(* POU FB_BACnet_AnalogOutput_EX, ST *)
FUNCTION_BLOCK FB_BACnet_AnalogOutput_EX
VAR_INPUT
	bEnablePV			: BOOL; (* enable present value with priority x in priority array, FALSE = priority x disable *)
	bNullPV				: BOOL; (* clear priority entry *)
	fPV					: REAL; (* decimal number for priority x, when input bEnablePV is TRUE *)
END_VAR
VAR_IN_OUT
	Device				: FB_BACnet_Device;
END_VAR
VAR_OUTPUT
	bReady				: BOOL;
	fPresentValue		: REAL;
	bOverridden			: BOOL;
	bOutOfService		: BOOL;
	bFault				: BOOL;
	bInAlarm			: BOOL;
	bNoOutput			: BOOL;
	bOpenLoop			: BOOL;
	bShortedLoop		: BOOL;
	bOtherFault			: BOOL;
	eEventState			: E_BACNETEVENTSTATE;
	bAckedTrans_ToOffNormal : BOOL;
	bAckedTrans_ToFault		: BOOL;
	bAckedTrans_ToNormal	: BOOL;
	nActivePrio			: UINT;
	tObjectID			: T_BACnet_ObjectIdentifier := 16#FFFFFFFF;
	bError				: BOOL;
	nErrorId			: UINT;
END_VAR
VAR
	_PresentValue AT%I*: REAL; 			(* ~(BACnet_PresentValue 			:		: )
								   			(BACnet_ObjectType 				: AO	: )	*)
    _PresentValue_Priority12 AT%Q*: DWORD;(* ~(BACnet_PresentValue_Priority12:		: )	*)
	_ActivePriority AT%I*: UDINT; 		(* ~(BACnet_ActivePriority 			:		: )	*)
	_ObjectId AT%I*: DWORD;				(* ~(BACnet_ObjectIdentifier		:		: LINK) *)
	_StatusFlags AT%I*: WORD; 			(* ~(BACnet_StatusFlags 			:		: )	*)
	_EventState AT%I*: WORD;			(* ~(BACnet_EventState 				:		: )	*)
	_Reliability AT%I*: WORD; 			(* ~(BACnet_Reliability 			:		: )	*)
	_AckedTransitions AT%I*:WORD;		(* ~(BACnet_AckedTransitions		:		: ) *)
	_StatusFlagsBits : ST_BACnet_StatusFlags;
	_AckedTransBits : ST_BACnet_EventTransitionBits;
	_nUpdateCount : UDINT := 0;
END_VAR
(* update server device *)
IF (Device._nUpdateCount = _nUpdateCount) THEN
	Device();
END_IF
(* remind current number of update counter *)
_nUpdateCount := Device._nUpdateCount;

IF Device.bFirstCycle THEN
	(* first call of the server device since reboot/reset *)
	bReady := FALSE;
	_PresentValue_Priority12 := F_BACnet_RealNothing();

ELSIF (F_BACnet_GetObjType(_ObjectId) <> BACnetObjectType_AnalogOutput) THEN
	(* wrong mapping / invalid object ID *)
	IF _ObjectId = 0 THEN
		nErrorId := BACnet_ERR_WRONG_MAPPING;
	ELSE
		nErrorId := BACnet_ERR_INVALID_OBJECTID;
	END_IF
	bReady := FALSE;

ELSIF (_StatusFlags < 4) THEN
	(* wrong mapping *)
	nErrorId := BACnet_ERR_WRONG_MAPPING;
	bReady := FALSE;

ELSIF Device.bOperational THEN
	(* ready state *)
	bReady := TRUE;
	nErrorId := BACnet_ERR_NO_ERROR;

	(* write into priority array *)
	_PresentValue_Priority12 := F_BACnet_RealPV(bEnablePV, bNullPV, fPV);

	(* present value *)
	fPresentValue := _PresentValue;

	(* build bit states *)
	_StatusFlagsBits := F_BACnet_StatusFlags(_StatusFlags);
	_AckedTransBits		:= F_BACnet_EventTransitionFlags(_AckedTransitions);

	(* copy states to output *)
	bOverridden := _StatusFlagsBits.overridden;
	bOutOfService := _StatusFlagsBits.out_of_service;
	bFault := _StatusFlagsBits.fault;
	bInAlarm := _StatusFlagsBits.in_alarm;
	bNoOutput := (_Reliability = BACnetReliability_no_output);
	bOpenLoop := (_Reliability = BACnetReliability_open_loop);
	bShortedLoop := (_Reliability = BACnetReliability_shorted_loop);
	bOtherFault := (_Reliability = BACnetReliability_unreliable_other);
	bAckedTrans_ToOffNormal := _AckedTransBits.to_offnormal;
	bAckedTrans_ToFault := _AckedTransBits.to_fault;
	bAckedTrans_ToNormal := _AckedTransBits.to_normal;
	tObjectID := _ObjectId;

	(* convert enumeration *)
	eEventState := _EventState;

	(* copy active priority *)
	nActivePrio := UDINT_TO_UINT(_ActivePriority);

ELSE
	(* server device not ready, reset local ready also *)
	bReady := FALSE;
	nErrorId := BACnet_ERR_OPERATIONAL;
END_IF
(* set error flag *)
bError := (nErrorId <> BACnet_ERR_NO_ERROR);
END_FUNCTION_BLOCK

(* POU FB_BACnet_AnalogOutput_RAW, ST *)
FUNCTION_BLOCK FB_BACnet_AnalogOutput_RAW
VAR_INPUT
	bEnablePV		: BOOL; (* enable present value with priority x in priority array, FALSE = priority x disable *)
	bNullPV			: BOOL; (* clear priority entry *)
	fPV				: REAL; (* decimal number for priority x, when input bEnablePV is TRUE *)
	bRawOverridden	AT%Q*: BOOL; (* ~(BACnet_RawIoStateOverride	:		: ) *)
	bNoOutput		: BOOL;
	bOpenLoop		: BOOL;
	bShortedLoop	: BOOL;
	bCommFailure	: BOOL;
	bOtherFault		: BOOL;
END_VAR
VAR_IN_OUT
	Device	: FB_BACnet_Device;
END_VAR
VAR_OUTPUT
	bReady			: BOOL;
	fPresentValue	: REAL;
	bOverridden		: BOOL;
	bOutOfService	: BOOL;
	bFault			: BOOL;
	bInAlarm		: BOOL;
	bAckedTrans_ToOffNormal : BOOL;
	bAckedTrans_ToFault		: BOOL;
	bAckedTrans_ToNormal	: BOOL;
	bError			: BOOL;
	nErrorId		: UINT;
	nRawOut			AT%I*: INT;			(* ~(BACnet_RawIoAnalogSignedValue : : ) *)
END_VAR
VAR
	_PresentValue AT%I*: REAL; 			(* ~(BACnet_PresentValue 			:		: )
								   			(BACnet_ObjectType 				: AO	: )	*)
	_ObjectId AT%I*: DWORD;				(* ~(BACnet_ObjectIdentifier		:		: LINK) *)
	_AckedTransitions AT%I*:WORD;		(* ~(BACnet_AckedTransitions		:		: ) *)
	_StatusFlags AT%I*: WORD; 			(* ~(BACnet_StatusFlags 			:		: )	*)
    _PresentValue_Priority12 AT%Q*: DWORD;(* ~(BACnet_PresentValue_Priority12:		: )	*)
	_Reliability AT%Q*: WORD := BACnetReliability_no_fault_detected;(* ~(BACnet_Reliability 	:		: )	*)
	_AckedTransBits : ST_BACnet_EventTransitionBits;
	_StatusFlagsBits : ST_BACnet_StatusFlags;
	_nUpdateCount : UDINT := 0;
END_VAR
(* update server device *)
IF (Device._nUpdateCount = _nUpdateCount) THEN
	Device();
END_IF
(* remind current number of update counter *)
_nUpdateCount := Device._nUpdateCount;

(* handle raw error *)
IF bNoOutput THEN
	_Reliability := BACnetReliability_no_output;
ELSIF bOpenLoop THEN
	_Reliability := BACnetReliability_open_loop;
ELSIF bShortedLoop THEN
	_Reliability := BACnetReliability_shorted_loop;
ELSIF bCommFailure THEN
	_Reliability := BACnetReliability_communication_failure;
ELSIF bOtherFault THEN
	_Reliability := BACnetReliability_unreliable_other;
ELSE
	_Reliability := BACnetReliability_no_fault_detected;
END_IF

IF Device.bFirstCycle THEN
	(* first call of the server device since reboot/reset *)
	bReady := FALSE;
	_PresentValue_Priority12 := F_BACnet_RealNothing();

ELSIF (_StatusFlags < 4) THEN
	(* wrong mapping *)
	nErrorId := BACnet_ERR_WRONG_MAPPING;
	bReady := FALSE;

ELSIF Device.bOperational THEN
	(* ready state *)
	bReady := TRUE;
	nErrorId := BACnet_ERR_NO_ERROR;

	(* write into priority array *)
	_PresentValue_Priority12 := F_BACnet_RealPV(bEnablePV, bNullPV, fPV);

	(* present value *)
	fPresentValue := _PresentValue;

	(* build bit states *)
	_StatusFlagsBits := F_BACnet_StatusFlags(_StatusFlags);
	_AckedTransBits		:= F_BACnet_EventTransitionFlags(_AckedTransitions);

	(* copy states to output *)
	bOverridden := _StatusFlagsBits.overridden;
	bOutOfService := _StatusFlagsBits.out_of_service;
	bFault := _StatusFlagsBits.fault;
	bInAlarm := _StatusFlagsBits.in_alarm;
	bAckedTrans_ToOffNormal := _AckedTransBits.to_offnormal;
	bAckedTrans_ToFault := _AckedTransBits.to_fault;
	bAckedTrans_ToNormal := _AckedTransBits.to_normal;

ELSE
	(* server device not ready, reset local ready also *)
	bReady := FALSE;
	nErrorId := BACnet_ERR_OPERATIONAL;
END_IF
(* set error flag *)
bError := (nErrorId <> BACnet_ERR_NO_ERROR);
END_FUNCTION_BLOCK

(* POU FB_BACnet_AnalogValue, ST *)
FUNCTION_BLOCK FB_BACnet_AnalogValue
VAR_INPUT
	bEnablePV		: BOOL; (* enable present value with priority x in priority array, FALSE = priority x disable *)
	bNullPV			: BOOL; (* clear priority entry *)
	fPV				: REAL; (* decimal number for priority x, when input bEnablePV is TRUE *)
END_VAR
VAR_IN_OUT
	Device			: FB_BACnet_Device;
END_VAR
VAR_OUTPUT
	bReady			: BOOL;
	fPresentValue	: REAL;
	bOverridden		: BOOL;
	bOutOfService	: BOOL;
	bFault			: BOOL;
	bInAlarm		: BOOL;
	bError			: BOOL;
	nErrorId		: UINT;
END_VAR
VAR
	_PresentValue AT%I*: REAL; 			(* ~(BACnet_PresentValue 			:		: )
								   			(BACnet_ObjectType 				: AV	: )	*)
    _PresentValue_Priority12 AT%Q*: DWORD;(* ~(BACnet_PresentValue_Priority12:		: )	*)
	_StatusFlags AT%I*: WORD; 			(* ~(BACnet_StatusFlags 			:		: )	*)
	_StatusFlagsBits : ST_BACnet_StatusFlags;
	_nUpdateCount : UDINT := 0;
END_VAR
(* update server device *)
IF (Device._nUpdateCount = _nUpdateCount) THEN
	Device();
END_IF
(* remind current number of update counter *)
_nUpdateCount := Device._nUpdateCount;

IF Device.bFirstCycle THEN
	(* first call of the server device since reboot/reset *)
	bReady := FALSE;
	_PresentValue_Priority12 := F_BACnet_RealNothing();
ELSIF (_StatusFlags < 4) THEN
	(* wrong mapping *)
	nErrorId := BACnet_ERR_WRONG_MAPPING;
	bReady := FALSE;

ELSIF Device.bOperational THEN
	(* ready state *)
	bReady := TRUE;
	nErrorId := BACnet_ERR_NO_ERROR;

	(* write into priority array *)
	_PresentValue_Priority12 := F_BACnet_RealPV(bEnablePV, bNullPV, fPV);

	(* present value *)
	fPresentValue := _PresentValue;

	(* build bit states *)
	_StatusFlagsBits := F_BACnet_StatusFlags(_StatusFlags);

	(* copy states to output *)
	bOverridden := _StatusFlagsBits.overridden;
	bOutOfService := _StatusFlagsBits.out_of_service;
	bFault := _StatusFlagsBits.fault;
	bInAlarm := _StatusFlagsBits.in_alarm;

ELSE
	(* server device not ready, reset local ready also *)
	bReady := FALSE;
	nErrorId := BACnet_ERR_OPERATIONAL;
END_IF
(* set error flag *)
bError := (nErrorId <> BACnet_ERR_NO_ERROR);
END_FUNCTION_BLOCK

(* POU FB_BACnet_AnalogValue_ADS, ST *)
FUNCTION_BLOCK FB_BACnet_AnalogValue_ADS
VAR_INPUT
	bEnablePV			: BOOL; (* enable PV write commands *)
	bNullPV				: BOOL; (* clear priority entry *)
	fPV					: REAL; (* decimal number for priority x, when input bEnablePV is TRUE and bNullPV is FALSE *)
	bManual				: BOOL; (* FALSE --> TRUE: write present_value immediately, FALSE: only write present_value on-change, TRUE: write present_value on-change and when device turns operational *)
	ePriority			: E_BACNETPRIORITY := BACNETPRIORITY_12;
END_VAR
VAR_IN_OUT
	Device				: FB_BACnet_Device;
END_VAR
VAR_OUTPUT
	bReady				: BOOL;
	bPvDone				: BOOL; (* present_value written over ADS *)
	fPresentValue		: REAL;
	bOverridden			: BOOL;
	bOutOfService		: BOOL;
	bFault				: BOOL;
	bInAlarm			: BOOL;
	tObjectID			: T_BACnet_ObjectIdentifier := 16#FFFFFFFF;
	bError				: BOOL;
	nErrorId			: UINT;
	nAdsErrorId			: UDINT;
END_VAR
VAR
	_PresentValue AT%I*: REAL; 			(* ~(BACnet_PresentValue 		:		: )
								   			(BACnet_ObjectType 			: AV	: )	*)
	_ObjectId AT%I*: DWORD;				(* ~(BACnet_ObjectIdentifier	:		: LINK) *)
	_StatusFlags AT%I*: WORD; 			(* ~(BACnet_StatusFlags 		:		: )	*)
    _PresentValue_Ads : DWORD;
	_StatusFlagsBits : ST_BACnet_StatusFlags;
	_nUpdateCount : UDINT := 0;
	_WriteProp : FB_BACnet_WriteProp;
	_rtrigManual : R_TRIG;
	_bNullPvOld : BOOL;
	_nObjType : E_BACNETOBJECTTYPE;
END_VAR
(* update server device *)
IF (Device._nUpdateCount = _nUpdateCount) THEN
	Device();
END_IF
(* remind current number of update counter *)
_nUpdateCount := Device._nUpdateCount;

(* trigger on manual flag *)
_rtrigManual(CLK:= bManual, Q=> );

(* decode object type *)
_nObjType := F_BACnet_GetObjType(_ObjectId);

IF Device.bFirstCycle THEN
	(* first call of the server device since reboot/reset *)
	bReady := FALSE;
	bPvDone := FALSE;

ELSIF _nObjType <> BACnetObjectType_AnalogValue THEN
	(* wrong mapped object type *)
	nErrorId := BACnet_ERR_INVALID_OBJECTTYPE;
	bReady := FALSE;
	bPvDone := FALSE;

ELSIF (_StatusFlags < 4) THEN
	(* wrong mapping *)
	nErrorId := BACnet_ERR_WRONG_MAPPING;
	bReady := FALSE;
	bPvDone := FALSE;

ELSIF Device.bOperational THEN

	IF Device.stAdsConn.bValid THEN
		(* write present_value on manual trigger, on-change and on operational recover *)
		IF		bEnablePV
			AND	(		_rtrigManual.Q
					OR	(MEMCMP(pBuf1:=ADR(fPV), pBuf2:=ADR(_PresentValue_Ads), n:=SIZEOF(_PresentValue_Ads)) <> 0)
					OR	((NOT bReady) AND bManual)
					OR	(bNullPV <> _bNullPvOld)
				)
		THEN
			_WriteProp.bExecute := TRUE;
			bPvDone := FALSE;
			(* write depending on enable state *)
			_PresentValue_Ads := F_BACnet_RealPV(TRUE, bNullPV, fPV);
			(* remind null flag *)
			_bNullPvOld := bNullPV;
		END_IF

		(* ready state *)
		IF (nAdsErrorId = 0) THEN
			bReady := TRUE;
			nErrorId := BACnet_ERR_NO_ERROR;
		END_IF

	ELSE
		(* invalid ADS connection *)
		bReady := FALSE;
		nErrorId := BACnet_ERR_INVALID_ADS_CONN;
		bPvDone := FALSE;
	END_IF

	(* present value *)
	fPresentValue := _PresentValue;

	(* build bit states *)
	_StatusFlagsBits := F_BACnet_StatusFlags(_StatusFlags);

	(* copy states to output *)
	bOverridden := _StatusFlagsBits.overridden;
	bOutOfService := _StatusFlagsBits.out_of_service;
	bFault := _StatusFlagsBits.fault;
	bInAlarm := _StatusFlagsBits.in_alarm;
	tObjectID := _ObjectId;

ELSE
	(* server device not ready, reset local ready also *)
	bReady := FALSE;
	nErrorId := BACnet_ERR_OPERATIONAL;
	bPvDone := FALSE;
END_IF

(* call write property command *)
_WriteProp(
	BACnetDevicePort	:= Device.stAdsConn.nAmsPort,
	bExecute			:= ,
	sNetId				:= Device.stAdsConn.sAmsNetId,
	ObjectType			:= _nObjType,
	PropertyID			:= BACnetPropertyIdentifier_PresentValue,
	Priority			:= ePriority,
	DataType			:= BACnetDataType_Real,
	ObjectInstance		:= F_BACnet_GetObjInstance(_ObjectId),
	ptrValue			:= ADR(_PresentValue_Ads),
	nLenValue			:= SIZEOF(_PresentValue_Ads),
	bDone				=> ,
	bBusy				=> ,
	bError				=> ,
	nErrID				=> );

(* set done flag *)
IF _WriteProp.bExecute AND (NOT _WriteProp.bBusy) THEN
	(* check if command was finished with error *)
	IF _WriteProp.bError THEN
		bPvDone		:= FALSE;
		bReady		:= FALSE;
		nErrorId	:= BACnet_ERR_ADS_Write;
	ELSE
		(* successful written *)
		bPvDone		:= TRUE;
	END_IF
	nAdsErrorId := _WriteProp.nErrID;
	(* reset execution bit *)
	_WriteProp(bExecute := FALSE);
END_IF

(* set error flag *)
bError := (nErrorId <> BACnet_ERR_NO_ERROR) OR (nAdsErrorId <> 0);
END_FUNCTION_BLOCK

(* POU FB_BACnet_AnalogValue_EX, ST *)
FUNCTION_BLOCK FB_BACnet_AnalogValue_EX
VAR_INPUT
	bEnablePV			: BOOL; (* enable present value with priority x in priority array, FALSE = priority x disable *)
	bNullPV				: BOOL; (* clear priority entry *)
	fPV					: REAL; (* decimal number for priority x, when input bEnablePV is TRUE *)
END_VAR
VAR_IN_OUT
	Device				: FB_BACnet_Device;
END_VAR
VAR_OUTPUT
	bReady				: BOOL;
	fPresentValue		: REAL;
	bOverridden			: BOOL;
	bOutOfService		: BOOL;
	bFault				: BOOL;
	bInAlarm			: BOOL;
	bOverRange			: BOOL;
	bUnderRange			: BOOL;
	bOtherFault			: BOOL;
	eEventState			: E_BACNETEVENTSTATE;
	bAckedTrans_ToOffNormal : BOOL;
	bAckedTrans_ToFault		: BOOL;
	bAckedTrans_ToNormal	: BOOL;
	nActivePrio			: UINT;
	tObjectID			: T_BACnet_ObjectIdentifier := 16#FFFFFFFF;
	bError				: BOOL;
	nErrorId			: UINT;
END_VAR
VAR
	_PresentValue AT%I*: REAL; 			(* ~(BACnet_PresentValue 				:		: )
								   			(BACnet_ObjectType 					: AV	: )	*)
    _PresentValue_Priority12 AT%Q*: DWORD;(* ~(BACnet_PresentValue_Priority12	:		: )	*)
	_ActivePriority AT%I*: UDINT; 		(* ~(BACnet_ActivePriority 				:		: )	*)
	_ObjectId AT%I*: DWORD;				(* ~(BACnet_ObjectIdentifier			:		: LINK) *)
	_StatusFlags AT%I*: WORD; 			(* ~(BACnet_StatusFlags 				:		: )	*)
	_EventState AT%I*: WORD;			(* ~(BACnet_EventState 					:		: )	*)
	_Reliability AT%I*: WORD;			(* ~(BACnet_Reliability 				:		: )	*)
	_AckedTransitions AT%I*:WORD;		(* ~(BACnet_AckedTransitions			:		: ) *)
	_StatusFlagsBits : ST_BACnet_StatusFlags;
	_AckedTransBits : ST_BACnet_EventTransitionBits;
	_nUpdateCount : UDINT := 0;
END_VAR
(* update server device *)
IF (Device._nUpdateCount = _nUpdateCount) THEN
	Device();
END_IF
(* remind current number of update counter *)
_nUpdateCount := Device._nUpdateCount;

IF Device.bFirstCycle THEN
	(* first call of the server device since reboot/reset *)
	bReady := FALSE;
	_PresentValue_Priority12 := F_BACnet_RealNothing();

ELSIF (F_BACnet_GetObjType(_ObjectId) <> BACnetObjectType_AnalogValue) THEN
	(* wrong mapping / invalid object ID *)
	IF _ObjectId = 0 THEN
		nErrorId := BACnet_ERR_WRONG_MAPPING;
	ELSE
		nErrorId := BACnet_ERR_INVALID_OBJECTID;
	END_IF
	bReady := FALSE;

ELSIF (_StatusFlags < 4) THEN
	(* wrong mapping *)
	nErrorId := BACnet_ERR_WRONG_MAPPING;
	bReady := FALSE;

ELSIF Device.bOperational THEN
	(* ready state *)
	bReady := TRUE;
	nErrorId := BACnet_ERR_NO_ERROR;

	(* write into priority array *)
	_PresentValue_Priority12 := F_BACnet_RealPV(bEnablePV, bNullPV, fPV);

	(* present value *)
	fPresentValue := _PresentValue;

	(* build bit states *)
	_StatusFlagsBits := F_BACnet_StatusFlags(_StatusFlags);
	_AckedTransBits		:= F_BACnet_EventTransitionFlags(_AckedTransitions);

	(* copy states to output *)
	bOverridden := _StatusFlagsBits.overridden;
	bOutOfService := _StatusFlagsBits.out_of_service;
	bFault := _StatusFlagsBits.fault;
	bInAlarm := _StatusFlagsBits.in_alarm;
	bOverRange := (_Reliability = BACnetReliability_over_range);
	bUnderRange := (_Reliability = BACnetReliability_under_range);
	bOtherFault := (_Reliability = BACnetReliability_unreliable_other);
	bAckedTrans_ToOffNormal := _AckedTransBits.to_offnormal;
	bAckedTrans_ToFault := _AckedTransBits.to_fault;
	bAckedTrans_ToNormal := _AckedTransBits.to_normal;
	tObjectID := _ObjectId;

	(* convert enumeration *)
	eEventState := _EventState;

	(* copy active priority *)
	nActivePrio := UDINT_TO_UINT(_ActivePriority);
ELSE
	(* server device not ready, reset local ready also *)
	bReady := FALSE;
	nErrorId := BACnet_ERR_OPERATIONAL;
END_IF
(* set error flag *)
bError := (nErrorId <> BACnet_ERR_NO_ERROR);
END_FUNCTION_BLOCK

(* POU FB_BACnet_Averaging, ST *)
FUNCTION_BLOCK FB_BACnet_Averaging
VAR_IN_OUT
	Device			: FB_BACnet_Device;
END_VAR
VAR_OUTPUT
	bReady			: BOOL;
	fAverageValue	: REAL;
	fMaximumValue	: REAL;
	fMinimumValue	: REAL;
	nValidSamples	: UDINT;
	nWindowSamples	: UDINT;
	nWindowInterval	: UDINT; (* [s] *)
	bError			: BOOL;
	nErrorId		: UINT;
END_VAR
VAR
	_AverageValue AT%I*: REAL;			(* ~(BACnet_AverageValue	:		: )
											(BACnet_ObjectType 		: AVG	: ) *)
	_MaximumValue AT%I*: REAL;			(* ~(BACnet_MaximumValue	:		: ) *)
	_MinimumValue AT%I*: REAL;			(* ~(BACnet_MinimumValue	:		: ) *)
	_ValidSamples AT%I*: UDINT;			(* ~(BACnet_ValidSamples	:		: ) *)
	_WindowSamples AT%I*: UDINT;		(* ~(BACnet_WindowSamples	:		: ) *)
	_WindowInterval AT%I*: UDINT;		(* ~(BACnet_WindowInterval	:		: ) *)
	_nUpdateCount : UDINT := 0;
END_VAR
(* update server device *)
IF (Device._nUpdateCount = _nUpdateCount) THEN
	Device();
END_IF
(* remind current number of update counter *)
_nUpdateCount := Device._nUpdateCount;

IF Device.bFirstCycle THEN
	(* first call of the server device since reboot/reset *)
	bReady := FALSE;
ELSIF Device.bOperational THEN
	(* ready state *)
	bReady := TRUE;
	nErrorId := BACnet_ERR_NO_ERROR;

	(* present values *)
	fAverageValue	:= _AverageValue;
	fMaximumValue	:= _MaximumValue;
	fMinimumValue	:= _MinimumValue;
	nValidSamples	:= _ValidSamples;
	nWindowSamples	:= _WindowSamples;
	nWindowInterval	:= _WindowInterval;

ELSE
	(* server device not ready, reset local ready also *)
	bReady := FALSE;
	nErrorId := BACnet_ERR_OPERATIONAL;
END_IF
(* set error flag *)
bError := (nErrorId <> BACnet_ERR_NO_ERROR);
END_FUNCTION_BLOCK

(* POU FB_BACnet_Averaging_EX, ST *)
FUNCTION_BLOCK FB_BACnet_Averaging_EX
VAR_IN_OUT
	Device				: FB_BACnet_Device;
END_VAR
VAR_OUTPUT
	bReady				: BOOL;
	fAverageValue		: REAL;
	fMaximumValue		: REAL;
	fMinimumValue		: REAL;
	nValidSamples		: UDINT;
	nWindowSamples		: UDINT;
	nWindowInterval		: UDINT; (* [s] *)
	tObjectID			: T_BACnet_ObjectIdentifier := 16#FFFFFFFF;
	bError				: BOOL;
	nErrorId			: UINT;
END_VAR
VAR
	_AverageValue AT%I*: REAL;			(* ~(BACnet_AverageValue	:		: )
											(BACnet_ObjectType 		: AVG	: ) *)
	_MaximumValue AT%I*: REAL;			(* ~(BACnet_MaximumValue	:		: ) *)
	_MinimumValue AT%I*: REAL;			(* ~(BACnet_MinimumValue	:		: ) *)
	_ValidSamples AT%I*: UDINT;			(* ~(BACnet_ValidSamples	:		: ) *)
	_WindowSamples AT%I*: UDINT;		(* ~(BACnet_WindowSamples	:		: ) *)
	_WindowInterval AT%I*: UDINT;		(* ~(BACnet_WindowInterval	:		: ) *)
	_ObjectId AT%I*: DWORD;				(* ~(BACnet_ObjectIdentifier:		: LINK) *)
	_nUpdateCount : UDINT := 0;
END_VAR
(* update server device *)
IF (Device._nUpdateCount = _nUpdateCount) THEN
	Device();
END_IF
(* remind current number of update counter *)
_nUpdateCount := Device._nUpdateCount;

IF Device.bFirstCycle THEN
	(* first call of the server device since reboot/reset *)
	bReady := FALSE;

ELSIF (F_BACnet_GetObjType(_ObjectId) <> BACnetObjectType_Averaging) THEN
	(* wrong mapping / invalid object ID *)
	IF _ObjectId = 0 THEN
		nErrorId := BACnet_ERR_WRONG_MAPPING;
	ELSE
		nErrorId := BACnet_ERR_INVALID_OBJECTID;
	END_IF
	bReady := FALSE;
	tObjectID := 16#FFFFFFFF;

ELSIF Device.bOperational THEN
	(* ready state *)
	bReady := TRUE;
	nErrorId := BACnet_ERR_NO_ERROR;

	(* present values *)
	fAverageValue	:= _AverageValue;
	fMaximumValue	:= _MaximumValue;
	fMinimumValue	:= _MinimumValue;
	nValidSamples	:= _ValidSamples;
	nWindowSamples	:= _WindowSamples;
	nWindowInterval	:= _WindowInterval;

	(* other states *)
	tObjectID := _ObjectId;

ELSE
	(* server device not ready, reset local ready also *)
	bReady := FALSE;
	nErrorId := BACnet_ERR_OPERATIONAL;
END_IF
(* set error flag *)
bError := (nErrorId <> BACnet_ERR_NO_ERROR);
END_FUNCTION_BLOCK

(* POU FB_BACnet_BinaryInput, ST *)
FUNCTION_BLOCK FB_BACnet_BinaryInput
VAR_IN_OUT
	Device	: FB_BACnet_Device;
END_VAR
VAR_OUTPUT
	bReady			: BOOL;
	bPresentValue	: BOOL;
	bOverridden		: BOOL;
	bOutOfService	: BOOL;
	bFault			: BOOL;
	bInAlarm		: BOOL;
	bError			: BOOL;
	nErrorId		: UINT;
END_VAR
VAR
	_PresentValue AT%I*: WORD; 			(* ~(BACnet_PresentValue 		:		: )
											(BACnet_ObjectType			:BI    	: )	*)
	_StatusFlags AT%I*: WORD; 			(* ~(BACnet_StatusFlags 		:	    : )	*)
	_StatusFlagsBits : ST_BACnet_StatusFlags;
	_nUpdateCount : UDINT := 0;
END_VAR
(* update server device *)
IF (Device._nUpdateCount = _nUpdateCount) THEN
	Device();
END_IF
(* remind current number of update counter *)
_nUpdateCount := Device._nUpdateCount;

(* check BitString format of StatusFlags --> if StatusFlags are less than 4, object isn't linked correctly *)
IF (_StatusFlags < 4) THEN
	(* wrong mapping *)
	nErrorId := BACnet_ERR_WRONG_MAPPING;
	bReady := FALSE;

ELSIF Device.bOperational THEN
	(* ready state *)
	bReady := TRUE;
	nErrorId := BACnet_ERR_NO_ERROR;

	(* present value *)
	bPresentValue := F_BinPV_To_Bool(_PresentValue);

	(* build bit states *)
	_StatusFlagsBits := F_BACnet_StatusFlags(_StatusFlags);

	(* copy states to output *)
	bOverridden := _StatusFlagsBits.overridden;
	bOutOfService := _StatusFlagsBits.out_of_service;
	bFault := _StatusFlagsBits.fault;
	bInAlarm := _StatusFlagsBits.in_alarm;

ELSE
	bReady := FALSE;
	nErrorId := BACnet_ERR_OPERATIONAL;
END_IF
(* set error flag *)
bError := (nErrorId <> BACnet_ERR_NO_ERROR);
END_FUNCTION_BLOCK

(* POU FB_BACnet_BinaryInput_EX, ST *)
FUNCTION_BLOCK FB_BACnet_BinaryInput_EX
VAR_IN_OUT
	Device	: FB_BACnet_Device;
END_VAR
VAR_OUTPUT
	bReady				: BOOL;
	bPresentValue		: BOOL;
	bOverridden			: BOOL;
	bOutOfService		: BOOL;
	bFault				: BOOL;
	bInAlarm			: BOOL;
	bNoSensor			: BOOL;
	bOpenLoop			: BOOL;
	bShortedLoop		: BOOL;
	bOtherFault			: BOOL;
	eEventState			: E_BACNETEVENTSTATE;
	bAckedTrans_ToOffNormal : BOOL;
	bAckedTrans_ToFault		: BOOL;
	bAckedTrans_ToNormal	: BOOL;
	nChangeOfState		: UDINT;
	tObjectID			: T_BACnet_ObjectIdentifier := 16#FFFFFFFF;
	bError				: BOOL;
	nErrorId			: UINT;
END_VAR
VAR
	_ChangeOfStateCount AT%I*: UDINT;		(* ~(BACnet_ChangeOfStateCount	:		: ) *)
	_ObjectId AT%I*: DWORD;					(* ~(BACnet_ObjectIdentifier	:		: LINK) *)
	_PresentValue AT%I*: WORD; 				(* ~(BACnet_PresentValue 		:		: )
												(BACnet_ObjectType			:BI    	: )	*)
	_StatusFlags AT%I*: WORD; 				(* ~(BACnet_StatusFlags 		:	    : )	*)
	_EventState AT%I*: WORD; 				(* ~(BACnet_EventState 			:	    : )	*)
	_Reliability AT%I*: WORD; 				(* ~(BACnet_Reliability 		:		: )	*)
	_AckedTransitions AT%I*:WORD;			(* ~(BACnet_AckedTransitions	:		: ) *)
	_AckedTransBits : ST_BACnet_EventTransitionBits;
	_StatusFlagsBits : ST_BACnet_StatusFlags;
	_nUpdateCount : UDINT := 0;
END_VAR
(* update server device *)
IF (Device._nUpdateCount = _nUpdateCount) THEN
	Device();
END_IF
(* remind current number of update counter *)
_nUpdateCount := Device._nUpdateCount;

(* check object type *)
IF (F_BACnet_GetObjType(_ObjectId) <> BACnetObjectType_BinaryInput) THEN
	(* wrong mapping / invalid object ID *)
	IF _ObjectId = 0 THEN
		nErrorId := BACnet_ERR_WRONG_MAPPING;
	ELSE
		nErrorId := BACnet_ERR_INVALID_OBJECTID;
	END_IF
	bReady := FALSE;

ELSIF (_StatusFlags < 4) THEN
	(* wrong mapping *)
	nErrorId := BACnet_ERR_WRONG_MAPPING;
	bReady := FALSE;

ELSIF Device.bOperational THEN
	(* ready state *)
	bReady := TRUE;
	nErrorId := BACnet_ERR_NO_ERROR;

	(* present value *)
	bPresentValue := F_BinPV_To_Bool(_PresentValue);

	(* build bit states *)
	_StatusFlagsBits := F_BACnet_StatusFlags(_StatusFlags);
	_AckedTransBits		:= F_BACnet_EventTransitionFlags(_AckedTransitions);

	(* copy states to output *)
	bOverridden := _StatusFlagsBits.overridden;
	bOutOfService := _StatusFlagsBits.out_of_service;
	bFault := _StatusFlagsBits.fault;
	bInAlarm := _StatusFlagsBits.in_alarm;
	bNoSensor := (_Reliability = BACnetReliability_no_sensor);
	bOpenLoop := (_Reliability = BACnetReliability_open_loop);
	bShortedLoop := (_Reliability = BACnetReliability_shorted_loop);
	bOtherFault := (_Reliability = BACnetReliability_unreliable_other);
	bAckedTrans_ToOffNormal := _AckedTransBits.to_offnormal;
	bAckedTrans_ToFault := _AckedTransBits.to_fault;
	bAckedTrans_ToNormal := _AckedTransBits.to_normal;
	tObjectID := _ObjectId;

	(* convert enumeration *)
	eEventState := _EventState;

	(* copy change_of_state_count *)
	nChangeOfState := _ChangeOfStateCount;
ELSE
	bReady := FALSE;
	nErrorId := BACnet_ERR_OPERATIONAL;
END_IF
(* set error flag *)
bError := (nErrorId <> BACnet_ERR_NO_ERROR);
END_FUNCTION_BLOCK

(* POU FB_BACnet_BinaryInput_RAW, ST *)
FUNCTION_BLOCK FB_BACnet_BinaryInput_RAW
VAR_INPUT
	bRawIn			AT%Q*: BOOL; (* ~(BACnet_RawIoBinaryBoolValue : : ) *)
	bNoSensor		: BOOL;
	bOpenLoop		: BOOL;
	bShortedLoop	: BOOL;
	bCommFailure	: BOOL;
	bOtherFault		: BOOL;
END_VAR
VAR_IN_OUT
	Device	: FB_BACnet_Device;
END_VAR
VAR_OUTPUT
	bReady			: BOOL;
	bPresentValue	: BOOL;
	bOverridden		: BOOL;
	bOutOfService	: BOOL;
	bFault			: BOOL;
	bInAlarm		: BOOL;
	bAckedTrans_ToOffNormal : BOOL;
	bAckedTrans_ToFault		: BOOL;
	bAckedTrans_ToNormal	: BOOL;
	bError			: BOOL;
	nErrorId		: UINT;
END_VAR
VAR
	_Reliability AT%Q*: WORD := BACnetReliability_no_fault_detected;(* ~(BACnet_Reliability 	:		: )	*)
	_ObjectId AT%I*: DWORD;				(* ~(BACnet_ObjectIdentifier	:		: LINK) *)
	_PresentValue AT%I*: WORD; 			(* ~(BACnet_PresentValue 		:		: )
											(BACnet_ObjectType			:BI    	: )	*)
	_StatusFlags AT%I*: WORD; 			(* ~(BACnet_StatusFlags 		:	    : )	*)
	_AckedTransitions AT%I*:WORD;		(* ~(BACnet_AckedTransitions	:		: ) *)
	_AckedTransBits : ST_BACnet_EventTransitionBits;
	_StatusFlagsBits : ST_BACnet_StatusFlags;
	_nUpdateCount : UDINT := 0;
END_VAR
(* update server device *)
IF (Device._nUpdateCount = _nUpdateCount) THEN
	Device();
END_IF
(* remind current number of update counter *)
_nUpdateCount := Device._nUpdateCount;

(* handle raw error *)
IF bNoSensor THEN
	_Reliability := BACnetReliability_no_sensor;
ELSIF bOpenLoop THEN
	_Reliability := BACnetReliability_open_loop;
ELSIF bShortedLoop THEN
	_Reliability := BACnetReliability_shorted_loop;
ELSIF bCommFailure THEN
	_Reliability := BACnetReliability_communication_failure;
ELSIF bOtherFault THEN
	_Reliability := BACnetReliability_unreliable_other;
ELSE
	_Reliability := BACnetReliability_no_fault_detected;
END_IF

(* check BitString format of StatusFlags --> if StatusFlags are less than 4, object isn't linked correctly *)
IF (_StatusFlags < 4) THEN
	(* wrong mapping *)
	nErrorId := BACnet_ERR_WRONG_MAPPING;
	bReady := FALSE;

ELSIF Device.bOperational THEN
	(* ready state *)
	bReady := TRUE;
	nErrorId := BACnet_ERR_NO_ERROR;

	(* present value *)
	bPresentValue := F_BinPV_To_Bool(_PresentValue);

	(* build bit states *)
	_StatusFlagsBits := F_BACnet_StatusFlags(_StatusFlags);
	_AckedTransBits		:= F_BACnet_EventTransitionFlags(_AckedTransitions);

	(* copy states to output *)
	bOverridden := _StatusFlagsBits.overridden;
	bOutOfService := _StatusFlagsBits.out_of_service;
	bFault := _StatusFlagsBits.fault;
	bInAlarm := _StatusFlagsBits.in_alarm;
	bAckedTrans_ToOffNormal := _AckedTransBits.to_offnormal;
	bAckedTrans_ToFault := _AckedTransBits.to_fault;
	bAckedTrans_ToNormal := _AckedTransBits.to_normal;

ELSE
	bReady := FALSE;
	nErrorId := BACnet_ERR_OPERATIONAL;
END_IF
(* set error flag *)
bError := (nErrorId <> BACnet_ERR_NO_ERROR);
END_FUNCTION_BLOCK

(* POU FB_BACnet_BinaryOutput, ST *)
FUNCTION_BLOCK FB_BACnet_BinaryOutput
VAR_INPUT
	bEnablePV		: BOOL; (* enable present value with priority x in priority array, FALSE = priority x disable *)
	bNullPV			: BOOL; (* clear priority entry *)
	bPV				: BOOL; (* present value bool type *)
END_VAR
VAR_IN_OUT
	Device			: FB_BACnet_Device;
END_VAR
VAR_OUTPUT
	bReady			: BOOL;
	bPresentValue	: BOOL;
	bOverridden		: BOOL;
	bOutOfService	: BOOL;
	bFault			: BOOL;
	bInAlarm		: BOOL;
	bError			: BOOL;
	nErrorId		: UINT;
END_VAR
VAR
	_PresentValue AT%I*: WORD; 			(* ~(BACnet_PresentValue 			:		: )
								   			(BACnet_ObjectType 				: BO	: )	*)
    _PresentValue_Priority12 AT%Q*: WORD;(* ~(BACnet_PresentValue_Priority12:		: )	*)
	_StatusFlags AT%I*: WORD; 			(* ~(BACnet_StatusFlags 			:		: )	*)
	_StatusFlagsBits : ST_BACnet_StatusFlags;
	_nUpdateCount : UDINT := 0;
END_VAR
(* update server device *)
IF (Device._nUpdateCount = _nUpdateCount) THEN
	Device();
END_IF
(* remind current number of update counter *)
_nUpdateCount := Device._nUpdateCount;

IF Device.bFirstCycle THEN
	(* first call of the server device since reboot/reset *)
	bReady := FALSE;
	_PresentValue_Priority12 := BACnetBinaryPV_Nothing;
ELSIF (_StatusFlags < 4) THEN
	(* wrong mapping *)
	nErrorId := BACnet_ERR_WRONG_MAPPING;
	bReady := FALSE;

ELSIF Device.bOperational THEN
	(* ready state *)
	bReady := TRUE;
	nErrorId := BACnet_ERR_NO_ERROR;

	(* write into priority array *)
	_PresentValue_Priority12 := F_Bool_To_BinPV(bEnablePV, bNullPV, bPV);

	(* present value *)
	bPresentValue := F_BinPV_To_Bool(_PresentValue);

	(* build bit states *)
	_StatusFlagsBits := F_BACnet_StatusFlags(_StatusFlags);

	(* copy states to output *)
	bOverridden := _StatusFlagsBits.overridden;
	bOutOfService := _StatusFlagsBits.out_of_service;
	bFault := _StatusFlagsBits.fault;
	bInAlarm := _StatusFlagsBits.in_alarm;

ELSE
	(* server device not ready, reset local ready also *)
	bReady := FALSE;
	nErrorId := BACnet_ERR_OPERATIONAL;
END_IF
(* set error flag *)
bError := (nErrorId <> BACnet_ERR_NO_ERROR);
END_FUNCTION_BLOCK

(* POU FB_BACnet_BinaryOutput_ADS, ST *)
FUNCTION_BLOCK FB_BACnet_BinaryOutput_ADS
VAR_INPUT
	bEnablePV			: BOOL; (* enable PV write commands *)
	bNullPV				: BOOL; (* clear priority entry *)
	bPV					: BOOL; (* present value bool type *)
	bManual				: BOOL; (* FALSE --> TRUE: write present_value immediately, FALSE: only write present_value on-change, TRUE: write present_value on-change and when device turns operational *)
	ePriority			: E_BACNETPRIORITY := BACNETPRIORITY_12;
END_VAR
VAR_IN_OUT
	Device				: FB_BACnet_Device;
END_VAR
VAR_OUTPUT
	bReady				: BOOL;
	bPvDone				: BOOL; (* present_value written over ADS *)
	bPresentValue		: BOOL;
	bOverridden			: BOOL;
	bOutOfService		: BOOL;
	bFault				: BOOL;
	bInAlarm			: BOOL;
	tObjectID			: T_BACnet_ObjectIdentifier := 16#FFFFFFFF;
	bError				: BOOL;
	nErrorId			: UINT;
	nAdsErrorId			: UDINT;
END_VAR
VAR
	_ObjectId AT%I*: DWORD;				(* ~(BACnet_ObjectIdentifier	:		: LINK) *)
	_PresentValue AT%I*: WORD; 			(* ~(BACnet_PresentValue 		:		: )
								   			(BACnet_ObjectType 			: BO	: )	*)
    _PresentValue_Ads : WORD;
	_StatusFlags AT%I*: WORD; 			(* ~(BACnet_StatusFlags 		:		: )	*)
	_StatusFlagsBits : ST_BACnet_StatusFlags;
	_nUpdateCount : UDINT := 0;
	_WriteProp : FB_BACnet_WriteProp;
	_rtrigManual : R_TRIG;
	_bNullPvOld : BOOL;
	_nObjType : E_BACNETOBJECTTYPE;
END_VAR
(* update server device *)
IF (Device._nUpdateCount = _nUpdateCount) THEN
	Device();
END_IF
(* remind current number of update counter *)
_nUpdateCount := Device._nUpdateCount;

(* trigger on manual flag *)
_rtrigManual(CLK:= bManual, Q=> );

(* decode object type *)
_nObjType := F_BACnet_GetObjType(_ObjectId);

IF Device.bFirstCycle THEN
	(* first call of the server device since reboot/reset *)
	bReady := FALSE;
	bPvDone := FALSE;

ELSIF _nObjType <> BACnetObjectType_BinaryOutput THEN
	(* wrong mapped object type *)
	nErrorId := BACnet_ERR_INVALID_OBJECTTYPE;
	bReady := FALSE;
	bPvDone := FALSE;

ELSIF (_StatusFlags < 4) THEN
	(* wrong mapping *)
	nErrorId := BACnet_ERR_WRONG_MAPPING;
	bReady := FALSE;
	bPvDone := FALSE;

ELSIF Device.bOperational THEN

	IF Device.stAdsConn.bValid THEN
		(* write present_value on manual trigger, on-change and on operational recover *)
		IF	(		bEnablePV
				AND	(		(bPV <> F_BinPV_To_Bool(_PresentValue_Ads))
						OR	((NOT bReady) AND bManual)
						OR	(bNullPV <> _bNullPvOld)
						OR	_rtrigManual.Q
					)
			)
		THEN
			_WriteProp.bExecute := TRUE;
			bPvDone := FALSE;
			(* write depending on enable state *)
			_PresentValue_Ads := F_Bool_To_BinPV(TRUE, bNullPV, bPV);
			_bNullPvOld := bNullPV;
		END_IF

		(* ready state *)
		IF (nAdsErrorId = 0) THEN
			bReady := TRUE;
			nErrorId := BACnet_ERR_NO_ERROR;
		END_IF

	ELSE
		(* invalid ADS connection *)
		bReady := FALSE;
		nErrorId := BACnet_ERR_INVALID_ADS_CONN;
		bPvDone := FALSE;
	END_IF


	(* present value *)
	bPresentValue := F_BinPV_To_Bool(_PresentValue);

	(* build bit states *)
	_StatusFlagsBits := F_BACnet_StatusFlags(_StatusFlags);

	(* copy states to output *)
	bOverridden := _StatusFlagsBits.overridden;
	bOutOfService := _StatusFlagsBits.out_of_service;
	bFault := _StatusFlagsBits.fault;
	bInAlarm := _StatusFlagsBits.in_alarm;
	tObjectID := _ObjectId;

ELSE
	(* server device not ready, reset local ready also *)
	bReady := FALSE;
	nErrorId := BACnet_ERR_OPERATIONAL;
	bPvDone := FALSE;
END_IF

(* call write property command *)
_WriteProp(
	BACnetDevicePort	:= Device.stAdsConn.nAmsPort,
	bExecute			:= ,
	sNetId				:= Device.stAdsConn.sAmsNetId,
	ObjectType			:= _nObjType,
	PropertyID			:= BACnetPropertyIdentifier_PresentValue,
	Priority			:= ePriority,
	DataType			:= BACnetDataType_BinaryPV,
	ObjectInstance		:= F_BACnet_GetObjInstance(_ObjectId),
	ptrValue			:= ADR(_PresentValue_Ads),
	nLenValue			:= SIZEOF(_PresentValue_Ads),
	bDone				=> ,
	bBusy				=> ,
	bError				=> ,
	nErrID				=> );

(* set done flag *)
IF _WriteProp.bExecute AND (NOT _WriteProp.bBusy) THEN
	(* check if command was finished with error *)
	IF _WriteProp.bError THEN
		bPvDone		:= FALSE;
		bReady		:= FALSE;
		nErrorId	:= BACnet_ERR_ADS_Write;
	ELSE
		(* successful written *)
		bPvDone		:= TRUE;
	END_IF
	nAdsErrorId := _WriteProp.nErrID;
	(* reset execution bit *)
	_WriteProp(bExecute := FALSE);
END_IF

(* set error flag *)
bError := (nErrorId <> BACnet_ERR_NO_ERROR) OR (nAdsErrorId <> 0);
END_FUNCTION_BLOCK

(* POU FB_BACnet_BinaryOutput_EX, ST *)
FUNCTION_BLOCK FB_BACnet_BinaryOutput_EX
VAR_INPUT
	bEnablePV			: BOOL; (* enable present value with priority x in priority array, FALSE = priority x disable *)
	bNullPV				: BOOL; (* clear priority entry *)
	bPV					: BOOL; (* present value bool type *)
END_VAR
VAR_IN_OUT
	Device				: FB_BACnet_Device;
END_VAR
VAR_OUTPUT
	bReady				: BOOL;
	bPresentValue		: BOOL;
	bOverridden			: BOOL;
	bOutOfService		: BOOL;
	bFault				: BOOL;
	bInAlarm			: BOOL;
	bNoOutput			: BOOL;
	bOpenLoop			: BOOL;
	bShortedLoop		: BOOL;
	bOtherFault			: BOOL;
	eEventState			: E_BACNETEVENTSTATE;
	bAckedTrans_ToOffNormal : BOOL;
	bAckedTrans_ToFault		: BOOL;
	bAckedTrans_ToNormal	: BOOL;
	nActivePrio			: UINT;
	nChangeOfState		: UDINT;
	tObjectID			: T_BACnet_ObjectIdentifier := 16#FFFFFFFF;
	bError				: BOOL;
	nErrorId			: UINT;
END_VAR
VAR_INPUT
END_VAR
VAR
	_ActivePriority AT%I*: UDINT; 		(* ~(BACnet_ActivePriority 			:		: )	*)
	_ChangeOfStateCount AT%I*: UDINT;	(* ~(BACnet_ChangeOfStateCount		:		: ) *)
	_ObjectId AT%I*: DWORD;				(* ~(BACnet_ObjectIdentifier		:		: LINK) *)
	_PresentValue AT%I*: WORD; 			(* ~(BACnet_PresentValue 			:		: )
								   			(BACnet_ObjectType 				: BO	: )	*)
    _PresentValue_Priority12 AT%Q*: WORD;(* ~(BACnet_PresentValue_Priority12:		: )	*)
	_StatusFlags AT%I*: WORD; 			(* ~(BACnet_StatusFlags 			:		: )	*)
	_EventState AT%I*: WORD; 			(* ~(BACnet_EventState 				:		: )	*)
	_Reliability AT%I*: WORD;			(* ~(BACnet_Reliability 			:		: )	*)
	_AckedTransitions AT%I*:WORD;		(* ~(BACnet_AckedTransitions		:		: ) *)
	_nUpdateCount : UDINT := 0;
	_AckedTransBits : ST_BACnet_EventTransitionBits;
	_StatusFlagsBits : ST_BACnet_StatusFlags;
END_VAR
(* update server device *)
IF (Device._nUpdateCount = _nUpdateCount) THEN
	Device();
END_IF
(* remind current number of update counter *)
_nUpdateCount := Device._nUpdateCount;

IF Device.bFirstCycle THEN
	(* first call of the server device since reboot/reset *)
	bReady := FALSE;
	_PresentValue_Priority12 := BACnetBinaryPV_Nothing;

ELSIF (F_BACnet_GetObjType(_ObjectId) <> BACnetObjectType_BinaryOutput) THEN
	(* wrong mapping / invalid object ID *)
	IF _ObjectId = 0 THEN
		nErrorId := BACnet_ERR_WRONG_MAPPING;
	ELSE
		nErrorId := BACnet_ERR_INVALID_OBJECTID;
	END_IF
	bReady := FALSE;

ELSIF (_StatusFlags < 4) THEN
	(* wrong mapping *)
	nErrorId := BACnet_ERR_WRONG_MAPPING;
	bReady := FALSE;

ELSIF Device.bOperational THEN
	(* ready state *)
	bReady := TRUE;
	nErrorId := BACnet_ERR_NO_ERROR;

	(* write into priority array *)
	_PresentValue_Priority12 := F_Bool_To_BinPV(bEnablePV, bNullPV, bPV);

	(* present value *)
	bPresentValue := F_BinPV_To_Bool(_PresentValue);

	(* build bit states *)
	_StatusFlagsBits := F_BACnet_StatusFlags(_StatusFlags);
	_AckedTransBits		:= F_BACnet_EventTransitionFlags(_AckedTransitions);

	(* copy states to output *)
	bOverridden := _StatusFlagsBits.overridden;
	bOutOfService := _StatusFlagsBits.out_of_service;
	bFault := _StatusFlagsBits.fault;
	bInAlarm := _StatusFlagsBits.in_alarm;
	bNoOutput := (_Reliability = BACnetReliability_no_output);
	bOpenLoop := (_Reliability = BACnetReliability_open_loop);
	bShortedLoop := (_Reliability = BACnetReliability_shorted_loop);
	bOtherFault := (_Reliability = BACnetReliability_unreliable_other);
	bAckedTrans_ToOffNormal := _AckedTransBits.to_offnormal;
	bAckedTrans_ToFault := _AckedTransBits.to_fault;
	bAckedTrans_ToNormal := _AckedTransBits.to_normal;
	tObjectID := _ObjectId;

	(* convert enumeration *)
	eEventState := _EventState;

	(* copy active priority *)
	nActivePrio := UDINT_TO_UINT(_ActivePriority);

	(* copy change_of_state_count *)
	nChangeOfState := _ChangeOfStateCount;
ELSE
	(* server device not ready, reset local ready also *)
	bReady := FALSE;
	nErrorId := BACnet_ERR_OPERATIONAL;
END_IF
(* set error flag *)
bError := (nErrorId <> BACnet_ERR_NO_ERROR);
END_FUNCTION_BLOCK

(* POU FB_BACnet_BinaryOutput_RAW, ST *)
FUNCTION_BLOCK FB_BACnet_BinaryOutput_RAW
VAR_INPUT
	bEnablePV		: BOOL; (* enable present value with priority x in priority array, FALSE = priority x disable *)
	bNullPV			: BOOL; (* clear priority entry *)
	bPV				: BOOL; (* present value bool type *)
	bFeedback		AT%Q*:BOOL;	(* ~(BACnet_FeedbackValue : : ) *)
	bRawOverridden	AT%Q*: BOOL; (* ~(BACnet_RawIoStateOverride	:		: ) *)
	bNoOutput		: BOOL;
	bOpenLoop		: BOOL;
	bShortedLoop	: BOOL;
	bCommFailure	: BOOL;
	bOtherFault		: BOOL;
END_VAR
VAR_IN_OUT
	Device		: FB_BACnet_Device;
END_VAR
VAR_OUTPUT
	bReady			: BOOL;
	bPresentValue	: BOOL;
	bOverridden		: BOOL;
	bOutOfService	: BOOL;
	bFault			: BOOL;
	bInAlarm		: BOOL;
	bAckedTrans_ToOffNormal : BOOL;
	bAckedTrans_ToFault		: BOOL;
	bAckedTrans_ToNormal	: BOOL;
	bError			: BOOL;
	nErrorId		: UINT;
	bRawOut			AT%I*: BOOL;			(* ~(BACnet_RawIoBinaryBoolValue	:		: ) *)
END_VAR
VAR
	_ObjectId AT%I*: DWORD;					(* ~(BACnet_ObjectIdentifier		:		: LINK) *)
	_PresentValue AT%I*: WORD; 				(* ~(BACnet_PresentValue 			:		: )
								   				(BACnet_ObjectType 				: BO	: )	*)
	_StatusFlags AT%I*: WORD; 				(* ~(BACnet_StatusFlags 			:		: )	*)
	_AckedTransitions AT%I*:WORD;			(* ~(BACnet_AckedTransitions		:		: ) *)
    _PresentValue_Priority12 AT%Q*: WORD;	(* ~(BACnet_PresentValue_Priority12	:		: )	*)
	_Reliability AT%Q*: WORD := BACnetReliability_no_fault_detected;(* ~(BACnet_Reliability 	:		: )	*)
	_AckedTransBits : ST_BACnet_EventTransitionBits;
	_StatusFlagsBits : ST_BACnet_StatusFlags;
	_nUpdateCount : UDINT := 0;
END_VAR
(* update server device *)
IF (Device._nUpdateCount = _nUpdateCount) THEN
	Device();
END_IF
(* remind current number of update counter *)
_nUpdateCount := Device._nUpdateCount;

(* handle raw error *)
IF bNoOutput THEN
	_Reliability := BACnetReliability_no_output;
ELSIF bOpenLoop THEN
	_Reliability := BACnetReliability_open_loop;
ELSIF bShortedLoop THEN
	_Reliability := BACnetReliability_shorted_loop;
ELSIF bCommFailure THEN
	_Reliability := BACnetReliability_communication_failure;
ELSIF bOtherFault THEN
	_Reliability := BACnetReliability_unreliable_other;
ELSE
	_Reliability := BACnetReliability_no_fault_detected;
END_IF

IF Device.bFirstCycle THEN
	(* first call of the server device since reboot/reset *)
	bReady := FALSE;
	_PresentValue_Priority12 := BACnetBinaryPV_Nothing;

ELSIF (_StatusFlags < 4) THEN
	(* wrong mapping *)
	nErrorId := BACnet_ERR_WRONG_MAPPING;
	bReady := FALSE;

ELSIF Device.bOperational THEN
	(* ready state *)
	bReady := TRUE;
	nErrorId := BACnet_ERR_NO_ERROR;

	(* write into priority array *)
	_PresentValue_Priority12 := F_Bool_To_BinPV(bEnablePV, bNullPV, bPV);

	(* present value *)
	bPresentValue := F_BinPV_To_Bool(_PresentValue);

	(* build bit states *)
	_StatusFlagsBits := F_BACnet_StatusFlags(_StatusFlags);
	_AckedTransBits		:= F_BACnet_EventTransitionFlags(_AckedTransitions);

	(* copy states to output *)
	bOverridden := _StatusFlagsBits.overridden;
	bOutOfService := _StatusFlagsBits.out_of_service;
	bFault := _StatusFlagsBits.fault;
	bInAlarm := _StatusFlagsBits.in_alarm;
	bAckedTrans_ToOffNormal := _AckedTransBits.to_offnormal;
	bAckedTrans_ToFault := _AckedTransBits.to_fault;
	bAckedTrans_ToNormal := _AckedTransBits.to_normal;

ELSE
	(* server device not ready, reset local ready also *)
	bReady := FALSE;
	nErrorId := BACnet_ERR_OPERATIONAL;
END_IF
(* set error flag *)
bError := (nErrorId <> BACnet_ERR_NO_ERROR);
END_FUNCTION_BLOCK

(* POU FB_BACnet_BinaryValue, ST *)
FUNCTION_BLOCK FB_BACnet_BinaryValue
VAR_INPUT
	bEnablePV		: BOOL; (* enable present value with priority x in priority array, FALSE = priority x disable *)
	bNullPV			: BOOL; (* clear priority entry *)
	bPV				: BOOL; (* present value bool type *)
END_VAR
VAR_IN_OUT
	Device			: FB_BACnet_Device;
END_VAR
VAR_OUTPUT
	bReady			: BOOL;
	bPresentValue	: BOOL;
	bOverridden		: BOOL;
	bOutOfService	: BOOL;
	bFault			: BOOL;
	bInAlarm		: BOOL;
	bError			: BOOL;
	nErrorId		: UINT;
END_VAR
VAR
	_PresentValue AT%I*: WORD; 			(* ~(BACnet_PresentValue 			:		: )
								   			(BACnet_ObjectType 				: BV	: )	*)
    _PresentValue_Priority12 AT%Q*: WORD;(* ~(BACnet_PresentValue_Priority12:		: )	*)
	_StatusFlags AT%I*: WORD; 			(* ~(BACnet_StatusFlags 			:		: )	*)
	_StatusFlagsBits : ST_BACnet_StatusFlags;
	_nUpdateCount : UDINT := 0;
END_VAR
(* update server device *)
IF (Device._nUpdateCount = _nUpdateCount) THEN
	Device();
END_IF
(* remind current number of update counter *)
_nUpdateCount := Device._nUpdateCount;

IF Device.bFirstCycle THEN
	(* first call of the server device since reboot/reset *)
	bReady := FALSE;
	_PresentValue_Priority12 := BACnetBinaryPV_Nothing;
ELSIF (_StatusFlags < 4) THEN
	(* wrong mapping *)
	nErrorId := BACnet_ERR_WRONG_MAPPING;
	bReady := FALSE;

ELSIF Device.bOperational THEN
	(* ready state *)
	bReady := TRUE;
	nErrorId := BACnet_ERR_NO_ERROR;

	(* write into priority array *)
	_PresentValue_Priority12 := F_Bool_To_BinPV(bEnablePV, bNullPV, bPV);

	(* present value *)
	bPresentValue := F_BinPV_To_Bool(_PresentValue);

	(* build bit states *)
	_StatusFlagsBits := F_BACnet_StatusFlags(_StatusFlags);

	(* copy states to output *)
	bOverridden := _StatusFlagsBits.overridden;
	bOutOfService := _StatusFlagsBits.out_of_service;
	bFault := _StatusFlagsBits.fault;
	bInAlarm := _StatusFlagsBits.in_alarm;

ELSE
	(* server device not ready, reset local ready also *)
	bReady := FALSE;
	nErrorId := BACnet_ERR_OPERATIONAL;
END_IF
(* set error flag *)
bError := (nErrorId <> BACnet_ERR_NO_ERROR);
END_FUNCTION_BLOCK

(* POU FB_BACnet_BinaryValue_ADS, ST *)
FUNCTION_BLOCK FB_BACnet_BinaryValue_ADS
VAR_INPUT
	bEnablePV			: BOOL; (* enable PV write commands *)
	bNullPV				: BOOL; (* clear priority entry *)
	bPV					: BOOL; (* present value bool type *)
	bManual				: BOOL; (* FALSE --> TRUE: write present_value immediately, FALSE: only write present_value on-change, TRUE: write present_value on-change and when device turns operational *)
	ePriority			: E_BACNETPRIORITY := BACNETPRIORITY_12;
END_VAR
VAR_IN_OUT
	Device				: FB_BACnet_Device;
END_VAR
VAR_OUTPUT
	bReady				: BOOL;
	bPvDone				: BOOL; (* present_value written over ADS *)
	bPresentValue		: BOOL;
	bOverridden			: BOOL;
	bOutOfService		: BOOL;
	bFault				: BOOL;
	bInAlarm			: BOOL;
	tObjectID			: T_BACnet_ObjectIdentifier := 16#FFFFFFFF;
	bError				: BOOL;
	nErrorId			: UINT;
	nAdsErrorId			: UDINT;
END_VAR
VAR
	_ObjectId AT%I*: DWORD;				(* ~(BACnet_ObjectIdentifier		:		: LINK) *)
	_PresentValue AT%I*: WORD; 			(* ~(BACnet_PresentValue 			:		: )
								   			(BACnet_ObjectType 				: BV	: )	*)
    _PresentValue_Ads : WORD;
	_StatusFlags AT%I*: WORD; 			(* ~(BACnet_StatusFlags 			:		: )	*)
	_StatusFlagsBits : ST_BACnet_StatusFlags;
	_nUpdateCount : UDINT := 0;
	_WriteProp : FB_BACnet_WriteProp;
	_rtrigManual : R_TRIG;
	_bNullPvOld : BOOL;
	_nObjType : E_BACNETOBJECTTYPE;
END_VAR
(* update server device *)
IF (Device._nUpdateCount = _nUpdateCount) THEN
	Device();
END_IF
(* remind current number of update counter *)
_nUpdateCount := Device._nUpdateCount;

(* trigger on manual flag *)
_rtrigManual(CLK:= bManual, Q=> );

(* decode object type *)
_nObjType := F_BACnet_GetObjType(_ObjectId);

IF Device.bFirstCycle THEN
	(* first call of the server device since reboot/reset *)
	bReady := FALSE;
	bPvDone := FALSE;

ELSIF _nObjType <> BACnetObjectType_BinaryValue THEN
	(* wrong mapped object type *)
	nErrorId := BACnet_ERR_INVALID_OBJECTTYPE;
	bReady := FALSE;
	bPvDone := FALSE;

ELSIF (_StatusFlags < 4) THEN
	(* wrong mapping *)
	nErrorId := BACnet_ERR_WRONG_MAPPING;
	bReady := FALSE;
	bPvDone := FALSE;

ELSIF Device.bOperational THEN

	IF Device.stAdsConn.bValid THEN
		(* write present_value on manual trigger, on-change and on operational recover *)
		IF (		bEnablePV
				AND	(		(bPV <> F_BinPV_To_Bool(_PresentValue_Ads))
						OR	((NOT bReady) AND bManual)
						OR	(bNullPV <> _bNullPvOld)
						OR	_rtrigManual.Q
					)
			)
		THEN
			_WriteProp.bExecute := TRUE;
			bPvDone := FALSE;
			(* write depending on enable state *)
			_PresentValue_Ads := F_Bool_To_BinPV(TRUE, bNullPV, bPV);
			_bNullPvOld := bNullPV;
		END_IF

		(* ready state *)
		IF (nAdsErrorId = 0) THEN
			bReady := TRUE;
			nErrorId := BACnet_ERR_NO_ERROR;
		END_IF

	ELSE
		(* invalid ADS connection *)
		bReady := FALSE;
		nErrorId := BACnet_ERR_INVALID_ADS_CONN;
		bPvDone := FALSE;
	END_IF

	(* present value *)
	bPresentValue := F_BinPV_To_Bool(_PresentValue);

	(* build bit states *)
	_StatusFlagsBits := F_BACnet_StatusFlags(_StatusFlags);

	(* copy states to output *)
	bOverridden := _StatusFlagsBits.overridden;
	bOutOfService := _StatusFlagsBits.out_of_service;
	bFault := _StatusFlagsBits.fault;
	bInAlarm := _StatusFlagsBits.in_alarm;
	tObjectID := _ObjectId;

ELSE
	(* server device not ready, reset local ready also *)
	bReady := FALSE;
	nErrorId := BACnet_ERR_OPERATIONAL;
	bPvDone := FALSE;
END_IF

(* call write property command *)
_WriteProp(
	BACnetDevicePort	:= Device.stAdsConn.nAmsPort,
	bExecute			:= ,
	sNetId				:= Device.stAdsConn.sAmsNetId,
	ObjectType			:= _nObjType,
	PropertyID			:= BACnetPropertyIdentifier_PresentValue,
	Priority			:= ePriority,
	DataType			:= BACnetDataType_BinaryPV,
	ObjectInstance		:= F_BACnet_GetObjInstance(_ObjectId),
	ptrValue			:= ADR(_PresentValue_Ads),
	nLenValue			:= SIZEOF(_PresentValue_Ads),
	bDone				=> ,
	bBusy				=> ,
	bError				=> ,
	nErrID				=> );

(* set done flag *)
IF _WriteProp.bExecute AND (NOT _WriteProp.bBusy) THEN
	(* check if command was finished with error *)
	IF _WriteProp.bError THEN
		bPvDone		:= FALSE;
		bReady		:= FALSE;
		nErrorId	:= BACnet_ERR_ADS_Write;
	ELSE
		(* successful written *)
		bPvDone		:= TRUE;
	END_IF
	nAdsErrorId := _WriteProp.nErrID;
	(* reset execution bit *)
	_WriteProp(bExecute := FALSE);
END_IF

(* set error flag *)
bError := (nErrorId <> BACnet_ERR_NO_ERROR) OR (nAdsErrorId <> 0);
END_FUNCTION_BLOCK

(* POU FB_BACnet_BinaryValue_EX, ST *)
FUNCTION_BLOCK FB_BACnet_BinaryValue_EX
VAR_INPUT
	bEnablePV			: BOOL; (* enable present value with priority x in priority array, FALSE = priority x disable *)
	bNullPV				: BOOL; (* clear priority entry *)
	bPV					: BOOL; (* present value bool type *)
END_VAR
VAR_IN_OUT
	Device				: FB_BACnet_Device;
END_VAR
VAR_OUTPUT
	bReady				: BOOL;
	bPresentValue		: BOOL;
	bOverridden			: BOOL;
	bOutOfService		: BOOL;
	bFault				: BOOL;
	bInAlarm			: BOOL;
	bOtherFault			: BOOL;
	eEventState			: E_BACNETEVENTSTATE;
	bAckedTrans_ToOffNormal : BOOL;
	bAckedTrans_ToFault		: BOOL;
	bAckedTrans_ToNormal	: BOOL;
	nActivePrio			: UINT;
	nChangeOfState		: UDINT;
	tObjectID			: T_BACnet_ObjectIdentifier := 16#FFFFFFFF;
	bError				: BOOL;
	nErrorId			: UINT;
END_VAR
VAR
	_ActivePriority AT%I*: UDINT; 		(* ~(BACnet_ActivePriority 			:		: )	*)
	_ChangeOfStateCount AT%I*: UDINT;	(* ~(BACnet_ChangeOfStateCount		:		: ) *)
	_ObjectId AT%I*: DWORD;				(* ~(BACnet_ObjectIdentifier		:		: LINK) *)
	_PresentValue AT%I*: WORD; 			(* ~(BACnet_PresentValue 			:		: )
								   			(BACnet_ObjectType 				: BV	: )	*)
    _PresentValue_Priority12 AT%Q*: WORD;(* ~(BACnet_PresentValue_Priority12:		: )	*)
	_StatusFlags AT%I*: WORD; 			(* ~(BACnet_StatusFlags 			:		: )	*)
	_EventState AT%I*: WORD; 			(* ~(BACnet_EventState 				:		: )	*)
	_Reliability AT%I*: WORD;			(* ~(BACnet_Reliability 			:		: )	*)
	_AckedTransitions AT%I*:WORD;		(* ~(BACnet_AckedTransitions:		: 		: ) *)
	_nUpdateCount : UDINT := 0;
	_AckedTransBits : ST_BACnet_EventTransitionBits;
	_StatusFlagsBits : ST_BACnet_StatusFlags;
END_VAR
(* update server device *)
IF (Device._nUpdateCount = _nUpdateCount) THEN
	Device();
END_IF
(* remind current number of update counter *)
_nUpdateCount := Device._nUpdateCount;

IF Device.bFirstCycle THEN
	(* first call of the server device since reboot/reset *)
	bReady := FALSE;
	_PresentValue_Priority12 := BACnetBinaryPV_Nothing;

ELSIF (F_BACnet_GetObjType(_ObjectId) <> BACnetObjectType_BinaryValue) THEN
	(* wrong mapping / invalid object ID *)
	IF _ObjectId = 0 THEN
		nErrorId := BACnet_ERR_WRONG_MAPPING;
	ELSE
		nErrorId := BACnet_ERR_INVALID_OBJECTID;
	END_IF
	bReady := FALSE;

ELSIF (_StatusFlags < 4) THEN
	(* wrong mapping *)
	nErrorId := BACnet_ERR_WRONG_MAPPING;
	bReady := FALSE;

ELSIF Device.bOperational THEN
	(* ready state *)
	bReady := TRUE;
	nErrorId := BACnet_ERR_NO_ERROR;

	(* write into priority array *)
	_PresentValue_Priority12 := F_Bool_To_BinPV(bEnablePV, bNullPV, bPV);

	(* present value *)
	bPresentValue := F_BinPV_To_Bool(_PresentValue);

	(* build bit states *)
	_StatusFlagsBits := F_BACnet_StatusFlags(_StatusFlags);
	_AckedTransBits		:= F_BACnet_EventTransitionFlags(_AckedTransitions);

	(* copy states to output *)
	bOverridden := _StatusFlagsBits.overridden;
	bOutOfService := _StatusFlagsBits.out_of_service;
	bFault := _StatusFlagsBits.fault;
	bInAlarm := _StatusFlagsBits.in_alarm;
	bOtherFault := (_Reliability = BACnetReliability_unreliable_other);
	bAckedTrans_ToOffNormal := _AckedTransBits.to_offnormal;
	bAckedTrans_ToFault := _AckedTransBits.to_fault;
	bAckedTrans_ToNormal := _AckedTransBits.to_normal;
	tObjectID := _ObjectId;

	(* convert enumeration *)
	eEventState := _EventState;

	(* copy active priority *)
	nActivePrio := UDINT_TO_UINT(_ActivePriority);

	(* copy change_of_state_count *)
	nChangeOfState := _ChangeOfStateCount;
ELSE
	(* server device not ready, reset local ready also *)
	bReady := FALSE;
	nErrorId := BACnet_ERR_OPERATIONAL;
END_IF
(* set error flag *)
bError := (nErrorId <> BACnet_ERR_NO_ERROR);
END_FUNCTION_BLOCK

(* POU FB_BACnet_Calendar, ST *)
FUNCTION_BLOCK FB_BACnet_Calendar
VAR_IN_OUT
	Device	: FB_BACnet_Device;
END_VAR
VAR_OUTPUT
	bReady			: BOOL;
	bPresentValue	: BOOL;
	bError			: BOOL;
	nErrorId		: UINT;
END_VAR
VAR
	_PresentValue AT%I*: BOOL;	(* ~(BACnet_PresentValue 			:		: )
									(BACnet_ObjectType 				: CAL	: )	*)
	_nUpdateCount : UDINT := 0;
END_VAR
(* update server device *)
IF (Device._nUpdateCount = _nUpdateCount) THEN
	Device();
END_IF
(* remind current number of update counter *)
_nUpdateCount := Device._nUpdateCount;

IF Device.bOperational THEN
	(* ready state *)
	bReady := TRUE;
	nErrorId := BACnet_ERR_NO_ERROR;
	(* present value *)
	bPresentValue := _PresentValue;
ELSE
	(* server device not ready, reset local ready also *)
	bReady := FALSE;
	nErrorId := BACnet_ERR_OPERATIONAL;
END_IF
(* set error flag *)
bError := (nErrorId <> BACnet_ERR_NO_ERROR);
END_FUNCTION_BLOCK

(* POU FB_BACnet_Calendar_EX, ST *)
FUNCTION_BLOCK FB_BACnet_Calendar_EX
VAR_IN_OUT
	Device				: FB_BACnet_Device;
END_VAR
VAR_OUTPUT
	bReady				: BOOL;
	bPresentValue		: BOOL;
	tObjectID			: T_BACnet_ObjectIdentifier := 16#FFFFFFFF;
	bError				: BOOL;
	nErrorId			: UINT;
END_VAR
VAR
	_ObjectId AT%I*: DWORD;		(* ~(BACnet_ObjectIdentifier:		: LINK) *)
	_PresentValue AT%I*: BOOL;	(* ~(BACnet_PresentValue 			:		: )
									(BACnet_ObjectType 				: CAL	: )	*)
	_nUpdateCount : UDINT := 0;
END_VAR
(* update server device *)
IF (Device._nUpdateCount = _nUpdateCount) THEN
	Device();
END_IF
(* remind current number of update counter *)
_nUpdateCount := Device._nUpdateCount;

IF (F_BACnet_GetObjType(_ObjectId) <> BACnetObjectType_Calendar) THEN
	(* wrong mapping / invalid object ID *)
	IF _ObjectId = 0 THEN
		nErrorId := BACnet_ERR_WRONG_MAPPING;
	ELSE
		nErrorId := BACnet_ERR_INVALID_OBJECTID;
	END_IF
	bReady := FALSE;
	tObjectID := 16#FFFFFFFF;

ELSIF Device.bOperational THEN
	(* ready state *)
	bReady := TRUE;
	nErrorId := BACnet_ERR_NO_ERROR;
	(* present value *)
	bPresentValue := _PresentValue;
	tObjectID := _ObjectId;
ELSE
	(* server device not ready, reset local ready also *)
	bReady := FALSE;
	nErrorId := BACnet_ERR_OPERATIONAL;
END_IF
(* set error flag *)
bError := (nErrorId <> BACnet_ERR_NO_ERROR);
END_FUNCTION_BLOCK

(* POU FB_BACnet_Command, ST *)
FUNCTION_BLOCK FB_BACnet_Command
VAR_INPUT
	bEnablePV		: BOOL;
	nPV				: UDINT;
	bRetrigger		: BOOL; (* execute selected action on raising edge again *)
END_VAR
VAR_IN_OUT
	Device	: FB_BACnet_Device;
END_VAR
VAR_OUTPUT
	bReady			: BOOL;
	nPresentValue	: UDINT;
	bAllWritesOk	: BOOL; (* all actions in selected action list are written *)
	bInProcess		: BOOL; (* object is busy *)
	bError			: BOOL;
	nErrorId		: UINT;
END_VAR
VAR
	_PresentValueIn AT%I*: UDINT; 		(* ~(BACnet_PresentValue 			:		: )
								   			(BACnet_ObjectType 				: CMD	: )	*)
    _PresentValueOut AT%Q*: UDINT;		(* ~(BACnet_PresentValue	 	   	:		: )	*)
	_InProcess AT%I*: BOOL;				(* ~(BACnet_InProcess 				:		: )	*)
	_AllWritesSuccessful AT%I*: BOOL;	(* ~(BACnet_AllWritesSuccessful		:		: )	*)
	_nUpdateCount : UDINT := 0;
	_rtrigRetriggerPv : R_TRIG;
	_bRetriggerReq : BOOL;
END_VAR
(* update server device *)
IF (Device._nUpdateCount = _nUpdateCount) THEN
	Device();
END_IF
(* remind current number of update counter *)
_nUpdateCount := Device._nUpdateCount;

(* call trigger *)
_rtrigRetriggerPv(CLK:= bRetrigger, Q=> );
IF _rtrigRetriggerPv.Q THEN
	_bRetriggerReq := TRUE;
END_IF

IF Device.bFirstCycle THEN
	(* first call of the server device since reboot/reset *)
	bReady := FALSE;
	_PresentValueOut := 0;
	_bRetriggerReq := FALSE;

ELSIF Device.bOperational THEN
	(* ready state *)
	bReady := TRUE;
	nErrorId := BACnet_ERR_NO_ERROR;
	(* activities *)
	bAllWritesOk := _AllWritesSuccessful;
	bInProcess := _InProcess;
	(* present value from BACnet *)
	nPresentValue := _PresentValueIn;
	(* present value to BACnet *)
	IF bEnablePV THEN
		IF (NOT bInProcess) THEN
			IF _bRetriggerReq THEN
				(* trigger action list *)
				_PresentValueOut := 0;
			ELSE
				(* set present value *)
				_PresentValueOut := nPV;
			END_IF
			_bRetriggerReq := FALSE;
		END_IF
	ELSE
		(* deactivate mapped present value --> other clients can write to property *)
		_PresentValueOut := 16#0;
		_bRetriggerReq := FALSE;
	END_IF
ELSE
	(* server device not ready, reset local ready also *)
	bReady := FALSE;
	nErrorId := BACnet_ERR_OPERATIONAL;
	_bRetriggerReq := FALSE;
END_IF
(* set error flag *)
bError := (nErrorId <> BACnet_ERR_NO_ERROR);
END_FUNCTION_BLOCK

(* POU FB_BACnet_Command_EX, ST *)
FUNCTION_BLOCK FB_BACnet_Command_EX
VAR_INPUT
	bEnablePV			: BOOL;
	nPV					: UDINT;
	bRetrigger			: BOOL; (* execute selected action on raising edge again *)
END_VAR
VAR_IN_OUT
	Device				: FB_BACnet_Device;
END_VAR
VAR_OUTPUT
	bReady				: BOOL;
	nPresentValue		: UDINT;
	bAllWritesOk		: BOOL; (* all actions in selected action list are written *)
	bInProcess			: BOOL; (* object is busy *)
	tObjectID			: T_BACnet_ObjectIdentifier := 16#FFFFFFFF;
	bError				: BOOL;
	nErrorId			: UINT;
END_VAR
VAR
	_PresentValueIn AT%I*: UDINT; 		(* ~(BACnet_PresentValue 			:		: )
								   			(BACnet_ObjectType 				: CMD	: )	*)
	_ObjectId AT%I*: DWORD;				(* ~(BACnet_ObjectIdentifier:		: LINK) *)
    _PresentValueOut AT%Q*: UDINT;		(* ~(BACnet_PresentValue	 	   	:		: )	*)
	_InProcess AT%I*: BOOL;				(* ~(BACnet_InProcess 				:		: )	*)
	_AllWritesSuccessful AT%I*: BOOL;	(* ~(BACnet_AllWritesSuccessful		:		: )	*)
	_nUpdateCount : UDINT := 0;
	_rtrigRetriggerPv : R_TRIG;
	_bRetriggerReq : BOOL;
END_VAR
(* update server device *)
IF (Device._nUpdateCount = _nUpdateCount) THEN
	Device();
END_IF
(* remind current number of update counter *)
_nUpdateCount := Device._nUpdateCount;

(* call trigger *)
_rtrigRetriggerPv(CLK:= bRetrigger, Q=> );
IF _rtrigRetriggerPv.Q THEN
	_bRetriggerReq := TRUE;
END_IF

IF Device.bFirstCycle THEN
	(* first call of the server device since reboot/reset *)
	bReady := FALSE;
	_PresentValueOut := 0;
	_bRetriggerReq := FALSE;

ELSIF (F_BACnet_GetObjType(_ObjectId) <> BACnetObjectType_Command) THEN
	(* wrong mapping / invalid object ID *)
	IF _ObjectId = 0 THEN
		nErrorId := BACnet_ERR_WRONG_MAPPING;
	ELSE
		nErrorId := BACnet_ERR_INVALID_OBJECTID;
	END_IF
	bReady := FALSE;
	tObjectID := 16#FFFFFFFF;
	_bRetriggerReq := FALSE;

ELSIF Device.bOperational THEN
	(* object ID *)
	tObjectID := _ObjectId;
	(* ready state *)
	bReady := TRUE;
	nErrorId := BACnet_ERR_NO_ERROR;
	(* activities *)
	bAllWritesOk := _AllWritesSuccessful;
	bInProcess := _InProcess;
	(* present value from BACnet *)
	nPresentValue := _PresentValueIn;
	(* present value to BACnet *)
	IF bEnablePV THEN
		IF (NOT bInProcess) THEN
			IF _bRetriggerReq THEN
				(* trigger action list *)
				_PresentValueOut := 0;
			ELSE
				(* set present value *)
				_PresentValueOut := nPV;
			END_IF
			_bRetriggerReq := FALSE;
		END_IF
	ELSE
		(* deactivate mapped present value --> other objects can write to property *)
		_PresentValueOut := 16#0;
		_bRetriggerReq := FALSE;
	END_IF
ELSE
	(* server device not ready, reset local ready also *)
	bReady := FALSE;
	nErrorId := BACnet_ERR_OPERATIONAL;
	_bRetriggerReq := FALSE;
END_IF
(* set error flag *)
bError := (nErrorId <> BACnet_ERR_NO_ERROR);
END_FUNCTION_BLOCK

(* POU FB_BACnet_DescriptionProperty, ST *)
FUNCTION_BLOCK FB_BACnet_DescriptionProperty
VAR_INPUT
	tObjectID			: T_BACnet_ObjectIdentifier := 16#FFFFFFFF;
	bAutoGet			: BOOL:=TRUE; (* TRUE = get data from property when ADS connection OR object ID changed *)
	bGet				: BOOL; (* FALSE --> TRUE = get data from property *)
END_VAR
VAR_IN_OUT
	stAdsConn			: ST_BACnet_AdsConnection;
END_VAR
VAR_OUTPUT
	bDone				: BOOL;
	bBusy				: BOOL;
	bError				: BOOL;
	nErrorId			: UINT;
	sText				: T_MaxString; (* Object description *)
END_VAR
VAR
	_fbReadProp		: FB_BACnet_ReadProp;
	_i				: INT;
	_rtrigGetSet	: R_TRIG;
	_nAdsReloadOld	: USINT;
	_tObjectIDOld	: T_BACnet_ObjectIdentifier := 16#FFFFFFFF;
	_StringExtDecode: FB_BACnet_StringExtDecode;
END_VAR
(* ADS read *)
_fbReadProp(
	BACnetDevicePort	:= stAdsConn.nAmsPort,
	bExecute			:= ,
	sNetId				:= stAdsConn.sAmsNetId,
	ObjectType			:= F_BACnet_GetObjType(tObjectID),
	PropertyID			:= BACnetPropertyIdentifier_Description,
	DataType			:= BACnetDataType_CharacterStringExt,
	ObjectInstance		:= F_BACnet_GetObjInstance(tObjectID),
	ptrValue			:= ADR(sText),
	nLenValue			:= SIZEOF(sText)-1,
	bDone				=> ,
	bBusy				=> ,
	bError				=> ,
	nErrID				=> ,
	nProcessedLen		=> );

(* trigger start event *)
_rtrigGetSet(CLK:= bGet, Q=> );

(* state machine *)
CASE _i OF

	0: (* Idle *)
		IF		(		(		_rtrigGetSet.Q
							OR	(_nAdsReloadOld <> stAdsConn.nReload)
							OR	(_tObjectIDOld <> tObjectID)
						)
					AND	bAutoGet
				)
			OR	_rtrigGetSet.Q
		THEN
			IF (NOT stAdsConn.bValid) THEN
				(* ADS connection not valid *)
				nErrorId := BACnet_ERR_INVALID_ADS_CONN;
			ELSIF (NOT stAdsConn.bServer AND NOT stAdsConn.bClient) THEN
				(* not a server nor a client *)
				nErrorId := BACnet_ERR_ADS_NoServerClient;
			ELSE
				nErrorId := BACnet_ERR_NO_ERROR;
				_i := 1;
				sText := '';
				(* remind ADS reload counter and parameter *)
				_nAdsReloadOld := stAdsConn.nReload;
				_tObjectIDOld := tObjectID;
			END_IF
			(* reset done flag *)
			bDone := FALSE;
		END_IF
		IF (NOT bGet) AND (NOT bAutoGet) THEN
			nErrorId := BACnet_ERR_NO_ERROR;
			bDone := FALSE;
		END_IF

	(* READ *)
	1: (* read object property data over ADS *)
		IF _fbReadProp.bExecute THEN
			IF _fbReadProp.bError THEN
				_i := 100;
				nErrorId := BACnet_ERR_ADS_Read;
				_fbReadProp.bExecute := FALSE;
			ELSIF (NOT _fbReadProp.bBusy) THEN
				_fbReadProp.bExecute := FALSE;
				(* decode property data *)
				_StringExtDecode(
					pChrStringExt	:= ADR(sText),
					cbOutSize		:= _fbReadProp.nProcessedLen,
					pOutString		:= ADR(sText),
					bValid			=> ,
					bOverflow		=> ,
					nLength			=> ,
					eSrcEncoding	=> );
				(* check overflow flag *)
				IF _StringExtDecode.bOverflow THEN
					nErrorId := BACnet_ERR_ADS_BufferSize;
				ELSIF (NOT _StringExtDecode.bValid) THEN
					nErrorId := BACnet_ERR_ADS_Encoding;
				END_IF
				(* DONE *)
				_i := 100;
			END_IF
		ELSE
			_fbReadProp.bExecute := TRUE;
		END_IF

	100: (* Done *)
		bDone := (nErrorId = BACnet_ERR_NO_ERROR);
		_i := 0;

END_CASE

(* set error flag *)
bError 	:= nErrorId > BACnet_ERR_NO_ERROR;
bBusy 	:= _i > 0;
END_FUNCTION_BLOCK

(* POU FB_BACnet_StringExtDecode, ST *)
FUNCTION_BLOCK FB_BACnet_StringExtDecode (* convert UTF-8/UCS2/UCS4/ISO8859-1 to Windows-1252 *)
VAR_INPUT
	pChrStringExt	: POINTER TO ST_BACnet_CharacterStringExt; (* BACnet character string data structure (header and string) *)
	pOutString		: POINTER TO T_MaxString; (* pointer to result buffer (Windows-1252 encoded) *)
	cbOutSize		: UDINT; (* byte size *)
END_VAR
VAR_OUTPUT
	bValid			: BOOL; (* Decoding successfull *)
	bOverflow		: BOOL; (* String length overflow (source string too long) *)
	bUnsupported	: BOOL; (* Souce encoding is unsupported (use ReadProp function and decode manually instead) *)
	nLength			: UDINT; (* out character length *)
	eSrcEncoding	: E_BACNETSTRINGENCODINGTYPES; (* input encoding *)
END_VAR
VAR_TEMP
	pText 			: POINTER TO BYTE;
	pByte			: POINTER TO BYTE;
END_VAR
(* preset valid to FALSE *)
bValid := FALSE;
bOverflow := FALSE;
bUnsupported := FALSE;
(* check pointer *)
IF (pChrStringExt = 0) OR (pOutString = 0) THEN
	nLength := 0;
(* check input size *)
ELSIF (cbOutSize = 0) THEN
	(* NULL string *)
	bValid := TRUE;
	pOutString^ := '';
	nLength := 0;
	eSrcEncoding := BACnetStringEncodingTypes_AnsiUtf8;
ELSE
	(* string data available *)
	IF (pChrStringExt^.cookie = 0) THEN
		(* new character string type *)
		nLength			:= UDINT_TO_UINT(pChrStringExt^.strLen);
		eSrcEncoding	:= UDINT_TO_INT(pChrStringExt^.encoding);
		pText			:= ADR(pChrStringExt^.stringData);
	ELSE
		(* ASCII/UTF-8 string *)
		nLength			:= _F_BACnet_ChrStrExtLen(pChrStringExt^);
		eSrcEncoding	:= BACnetStringEncodingTypes_AnsiUtf8;
		pText			:= pChrStringExt;
	END_IF

	(* check size *)
	IF (nLength = 0) THEN
		(* no data *)
		bValid := TRUE;
		pOutString^ := '';
	ELSIF (nLength <= cbOutSize) THEN
		(* copy to output buffer first *)
		MEMMOVE(destAddr:= pOutString, srcAddr:= pText, n:= nLength);

		(* decode and copy *)
		CASE eSrcEncoding OF

			BACnetStringEncodingTypes_AnsiUtf8:
				bValid := TRUE;
				nLength := UDINT_TO_UINT(_F_BACnet_DecodeUTF8(pOutString, nLength));

			BACnetStringEncodingTypes_UCS2:
				bValid := TRUE;
				nLength := UDINT_TO_UINT(_F_BACnet_DecodeUCS2(pOutString, nLength));

			BACnetStringEncodingTypes_UCS4:
				bValid := TRUE;
				nLength := UDINT_TO_UINT(_F_BACnet_DecodeUCS4(pOutString, nLength));

			BACnetStringEncodingTypes_ISO8859:
				bValid := TRUE;
				(* check if string termination is already part of string *)
				pByte := pOutString + nLength - 1;
				IF (pByte^ = 16#00) THEN
					(* termination already part of string *)
					nLength := nLength - 1;
				ELSE
					(* add string termination *)
					pByte := pOutString + nLength;
					pByte^ := 16#00;
				END_IF

			ELSE
				bUnsupported := TRUE;

		END_CASE
	ELSE
		(* text too long *)
		nLength := 0;
		pOutString^ := '';
		bOverflow := TRUE;
	END_IF
END_IF
END_FUNCTION_BLOCK

(* POU FB_BACnet_EventEnrollment, ST *)
FUNCTION_BLOCK FB_BACnet_EventEnrollment
VAR_IN_OUT
	Device					: FB_BACnet_Device;
END_VAR
VAR_OUTPUT
	bReady					: BOOL;
	eEventState				: E_BACNETEVENTSTATE;
	bAckedTrans_ToOffNormal : BOOL;
	bAckedTrans_ToFault		: BOOL;
	bAckedTrans_ToNormal	: BOOL;
	bError					: BOOL;
	nErrorId				: UINT;
END_VAR
VAR
	_EventState AT%I*: WORD; 			(* ~(BACnet_EventState 			:		: )
											(BACnet_ObjectType			: EE	: )	*)
	_AckedTransitions AT%I*: WORD; 		(* ~(BACnet_AckedTransitions 	:		: )	*)
	_AckedTransBits : ST_BACnet_EventTransitionBits;
	_nUpdateCount : UDINT := 0;
END_VAR
(* update server device *)
IF (Device._nUpdateCount = _nUpdateCount) THEN
	Device();
END_IF
(* remind current number of update counter *)
_nUpdateCount := Device._nUpdateCount;

(* check BitString format *)
IF (_AckedTransitions < 5) THEN
	(* wrong mapping *)
	nErrorId := BACnet_ERR_WRONG_MAPPING;
	bReady := FALSE;

ELSIF Device.bOperational THEN
	(* ready state *)
	bReady := TRUE;
	nErrorId := BACnet_ERR_NO_ERROR;

	(* copy states *)
	bAckedTrans_ToOffNormal := _AckedTransBits.to_offnormal;
	bAckedTrans_ToFault := _AckedTransBits.to_fault;
	bAckedTrans_ToNormal := _AckedTransBits.to_normal;
	eEventState := _EventState;

ELSE
	bReady := FALSE;
	nErrorId := BACnet_ERR_OPERATIONAL;
END_IF
(* set error flag *)
bError := (nErrorId <> BACnet_ERR_NO_ERROR);
END_FUNCTION_BLOCK

(* POU FB_BACnet_EventEnrollment_EX, ST *)
FUNCTION_BLOCK FB_BACnet_EventEnrollment_EX
VAR_IN_OUT
	Device				: FB_BACnet_Device;
END_VAR
VAR_OUTPUT
	bReady				: BOOL;
	eEventState			: E_BACNETEVENTSTATE;
	bEventEnable_ToOffNormal: BOOL;
	bEventEnable_ToFault: BOOL;
	bEventEnable_ToNormal: BOOL;
	bAckedTrans_ToOffNormal: BOOL;
	bAckedTrans_ToFault	: BOOL;
	bAckedTrans_ToNormal: BOOL;
	tObjectID			: T_BACnet_ObjectIdentifier := 16#FFFFFFFF;
	bError				: BOOL;
	nErrorId			: UINT;
END_VAR
VAR
	_ObjectId AT%I*: DWORD;			(* ~(BACnet_ObjectIdentifier	:		: LINK) *)
	_EventState AT%I*: WORD; 		(* ~(BACnet_EventState 			:		: )
										(BACnet_ObjectType			: EE	: )	*)
	_AckedTransitions AT%I*: WORD; 	(* ~(BACnet_AckedTransitions 	:		: )	*)
	_EventEnable AT%I*: WORD; 		(* ~(BACnet_EventEnable		 	:		: )	*)
	_EventTransBits : ST_BACnet_EventTransitionBits;
	_nUpdateCount : UDINT := 0;
END_VAR
(* update server device *)
IF (Device._nUpdateCount = _nUpdateCount) THEN
	Device();
END_IF
(* remind current number of update counter *)
_nUpdateCount := Device._nUpdateCount;

(* check BitString format *)
IF (F_BACnet_GetObjType(_ObjectId) <> BACnetObjectType_EventEnrollment) THEN
	(* wrong mapping / invalid object ID *)
	IF _ObjectId = 0 THEN
		nErrorId := BACnet_ERR_WRONG_MAPPING;
	ELSE
		nErrorId := BACnet_ERR_INVALID_OBJECTID;
	END_IF
	bReady := FALSE;
	tObjectID := 16#FFFFFFFF;

ELSIF (_AckedTransitions < 5) THEN
	(* wrong mapping *)
	nErrorId := BACnet_ERR_WRONG_MAPPING;
	bReady := FALSE;

ELSIF Device.bOperational THEN
	(* ready state *)
	bReady := TRUE;
	nErrorId := BACnet_ERR_NO_ERROR;

	(* copy states *)
	_EventTransBits			:= F_BACnet_EventTransitionFlags(_AckedTransitions);
	bAckedTrans_ToOffNormal	:= _EventTransBits.to_offnormal;
	bAckedTrans_ToFault		:= _EventTransBits.to_fault;
	bAckedTrans_ToNormal	:= _EventTransBits.to_normal;
	_EventTransBits			:= F_BACnet_EventTransitionFlags(_EventEnable);
	bEventEnable_ToOffNormal:= _EventTransBits.to_offnormal;
	bEventEnable_ToFault	:= _EventTransBits.to_fault;
	bEventEnable_ToNormal	:= _EventTransBits.to_normal;
	eEventState				:= _EventState;
	tObjectID			:= F_BACnet_GetObjInstance(_ObjectId);

ELSE
	bReady := FALSE;
	nErrorId := BACnet_ERR_OPERATIONAL;
END_IF
(* set error flag *)
bError := (nErrorId <> BACnet_ERR_NO_ERROR);
END_FUNCTION_BLOCK

(* POU FB_BACnet_EventLog, ST *)
FUNCTION_BLOCK FB_BACnet_EventLog
VAR_IN_OUT
	Device	: FB_BACnet_Device;
END_VAR
VAR_OUTPUT
	bReady			: BOOL;
	bLogEnable		: BOOL;
	nTotalCount		: UDINT;
	bError			: BOOL;
	nErrorId		: UINT;
END_VAR
VAR
	_TotalRecordCount AT%I*: UDINT;	(* ~(BACnet_TotalRecordCount:		: )
										(BACnet_ObjectType		: ELOG	: )	*)
	_LogEnable AT%I*: BOOL;			(* ~(BACnet_LogEnable		: 		: )	*)
	_nUpdateCount : UDINT := 0;
END_VAR
(* update server device *)
IF (Device._nUpdateCount = _nUpdateCount) THEN
	Device();
END_IF
(* remind current number of update counter *)
_nUpdateCount := Device._nUpdateCount;

IF Device.bOperational THEN
	(* ready state *)
	bReady := TRUE;
	nErrorId := BACnet_ERR_NO_ERROR;
	bLogEnable := _LogEnable;

	(* other states *)
	nTotalCount := _TotalRecordCount;

ELSE
	bReady := FALSE;
	nErrorId := BACnet_ERR_OPERATIONAL;
END_IF
(* set error flag *)
bError := (nErrorId <> BACnet_ERR_NO_ERROR);
END_FUNCTION_BLOCK

(* POU FB_BACnet_EventLog_EX, ST *)
FUNCTION_BLOCK FB_BACnet_EventLog_EX
VAR_IN_OUT
	Device	: FB_BACnet_Device;
END_VAR
VAR_OUTPUT
	bReady			: BOOL;
	bLogEnable		: BOOL;
	nRecordCount	: UDINT;
	nTotalCount		: UDINT;
	eEventState		: E_BACNETEVENTSTATE;
	bAckedTrans_ToOffNormal : BOOL;
	bAckedTrans_ToFault		: BOOL;
	bAckedTrans_ToNormal	: BOOL;
	tObjectID		: DINT := -1;
	bError			: BOOL;
	nErrorId		: UINT;
END_VAR
VAR
	_RecordCount AT%I*: UDINT;		(* ~(BACnet_RecordCount			:		: )
										(BACnet_ObjectType			: ELOG	: )	*)
	_TotalRecordCount AT%I*: UDINT;	(* ~(BACnet_TotalRecordCount	:		: )	*)
	_ObjectId AT%I*: DWORD;			(* ~(BACnet_ObjectIdentifier	:		: LINK) *)
	_EventState AT%I*: WORD;		(* ~(BACnet_EventState			:		: )	*)
	_AckedTransitions AT%I*:WORD;	(* ~(BACnet_AckedTransitions	:		: ) *)
	_LogEnable AT%I*: BOOL;			(* ~(BACnet_LogEnable			: 		: )	*)
	_AckedTransBits : ST_BACnet_EventTransitionBits;
	_nUpdateCount : UDINT := 0;
END_VAR
(* update server device *)
IF (Device._nUpdateCount = _nUpdateCount) THEN
	Device();
END_IF
(* remind current number of update counter *)
_nUpdateCount := Device._nUpdateCount;

(* check object type *)
IF (F_BACnet_GetObjType(_ObjectId) <> BACnetObjectType_EventLog) THEN
	(* wrong mapping / invalid object ID *)
	IF _ObjectId = 0 THEN
		nErrorId := BACnet_ERR_WRONG_MAPPING;
	ELSE
		nErrorId := BACnet_ERR_INVALID_OBJECTID;
	END_IF
	bReady := FALSE;

ELSIF Device.bOperational THEN
	(* ready state *)
	bReady := TRUE;
	bLogEnable := _LogEnable;
	nErrorId := BACnet_ERR_NO_ERROR;

	(* build bit states *)
	_AckedTransBits		:= F_BACnet_EventTransitionFlags(_AckedTransitions);
	bAckedTrans_ToOffNormal := _AckedTransBits.to_offnormal;
	bAckedTrans_ToFault := _AckedTransBits.to_fault;
	bAckedTrans_ToNormal := _AckedTransBits.to_normal;
	tObjectID := _ObjectId;

	(* convert enumeration *)
	eEventState := _EventState;

	(* other states *)
	nRecordCount := _RecordCount;
	nTotalCount := _TotalRecordCount;

ELSE
	bReady := FALSE;
	nErrorId := BACnet_ERR_OPERATIONAL;
END_IF
(* set error flag *)
bError := (nErrorId <> BACnet_ERR_NO_ERROR);
END_FUNCTION_BLOCK

(* POU FB_BACnet_EventMessageTextsProperty, ST *)
FUNCTION_BLOCK FB_BACnet_EventMessageTextsProperty
VAR_INPUT
	tObjectID			: T_BACnet_ObjectIdentifier := 16#FFFFFFFF;
	bAutoGet			: BOOL:=TRUE; (* TRUE = get data from property when ADS connection OR object ID changed *)
	bGet				: BOOL; (* FALSE --> TRUE = get data from property *)
END_VAR
VAR_IN_OUT
	stAdsConn			: ST_BACnet_AdsConnection;
END_VAR
VAR_OUTPUT
	bDone				: BOOL;
	bBusy				: BOOL;
	bError				: BOOL;
	nErrorId			: UINT;
	arrTexts			: ARRAY[0..2] OF T_MaxString; (* Windows-1252 encoded *)
END_VAR
VAR
	_fbReadProp		: FB_BACnet_ReadProp;
	_i				: INT;
	_rtrigGet		: R_TRIG;

	_iEntry			: INT;
	_pEntry			: POINTER TO ST_BACnet_CharacterStringExtListEntry;
	_pText			: POINTER TO BYTE;
	_pByte			: POINTER TO BYTE;
	_bNextEntry		: BOOL;
	_cbEntrySize	: UDINT;
	_cbTmpSize		: UDINT;
	_cbTotalBuf		: UDINT;
	_nAdsReloadOld	: USINT;
	_tObjectIDOld	: T_BACnet_ObjectIdentifier := 16#FFFFFFFF;
	_strExtDecode	: FB_BACnet_StringExtDecode;

END_VAR
(*

Listheader:

typedef struct _ListEntryHdr
{
      DWORD nEntrySize;
      DWORD hdrInfo;
}ListEntryHdr, *PListEntryHdr;


typedef struct _BACnetCharacterString
{
      ULONG       cookie            : 8; // = 0 -> do differentiate normal strings
      ULONG       encoding          : 8; 
      ULONG       strLen            : 16;
      BYTE        stringData[BACNET_STRING_MAXLENGTH];
}BACnetCharacterString, *PBACnetCharacterString;

#define     BACNET_STRING_MAXLENGTH 256

*)

(* ADS read *)
_fbReadProp(
	BACnetDevicePort	:= stAdsConn.nAmsPort,
	bExecute			:= ,
	sNetId				:= stAdsConn.sAmsNetId,
	ObjectType			:= F_BACnet_GetObjType(tObjectID),
	PropertyID			:= BACnetPropertyIdentifier_EventMessageTexts,
	DataType			:= BACnetDataType_CharacterStringExtList,
	ObjectInstance		:= F_BACnet_GetObjInstance(tObjectID),
	ptrValue			:= ADR(stBACnet_AdsBuffer.arrData),
	nLenValue			:= SIZEOF(stBACnet_AdsBuffer.arrData),
	bDone				=> ,
	bBusy				=> ,
	bError				=> ,
	nErrID				=> ,
	nProcessedLen		=> );

(* trigger start event *)
_rtrigGet(CLK:= bGet, Q=> );

(* state machine *)
CASE _i OF

	0: (* Idle *)
		IF 		_rtrigGet.Q
			OR	(		(		(_nAdsReloadOld <> stAdsConn.nReload)
							OR	(_tObjectIDOld <> tObjectID)
						)
					AND	bAutoGet
				)
		THEN
			IF (NOT stAdsConn.bValid) THEN
				(* ADS connection not valid *)
				nErrorId := BACnet_ERR_INVALID_ADS_CONN;
			ELSIF (NOT stAdsConn.bServer AND NOT stAdsConn.bClient) THEN
				(* not a server nor a client *)
				nErrorId := BACnet_ERR_ADS_NoServerClient;
			ELSE
				_i := 1;
				nErrorId := BACnet_ERR_NO_ERROR;
				(* remind parameter *)
				_tObjectIDOld := tObjectID;
				_nAdsReloadOld := stAdsConn.nReload;
			END_IF
			(* reset done flag *)
			bDone := FALSE;
		END_IF
		IF (NOT bGet) AND (NOT bAutoGet) THEN
			nErrorId := BACnet_ERR_NO_ERROR;
			bDone := FALSE;
		END_IF

	(* READ *)
	1: (* read object property data over ADS *)
		IF TestAndSet(stBACnet_AdsBuffer.bTestSet) THEN
			IF _fbReadProp.bExecute THEN
				IF _fbReadProp.bError THEN
					_i := 100;
					nErrorId := BACnet_ERR_ADS_Read;
					_fbReadProp.bExecute := FALSE;
				ELSIF (NOT _fbReadProp.bBusy) THEN
					_i := 2;
					_fbReadProp.bExecute := FALSE;
					_pEntry := ADR(stBACnet_AdsBuffer.arrData);
					MEMSET(ADR(arrTexts), 0, SIZEOF(arrTexts));
					_cbTotalBuf := 0;
					_iEntry := 0;
				END_IF
			ELSE
				(* lock global ADS buffer and start reading *)
				IF stBACnet_AdsBuffer.iLocked = 0 THEN
					_fbReadProp.bExecute := TRUE;
					stBACnet_AdsBuffer.iLocked := SIZEOF(stBACnet_AdsBuffer.arrData);
				END_IF
			END_IF

			(* release temporary task lock *)
			stBACnet_AdsBuffer.bTestSet := FALSE;
		END_IF

	2: (* select time value *)
		WHILE (_i = 2) DO
			_cbEntrySize := _pEntry^.nEntrySize AND 16#7FFFFFFF;
			(* check entry size *)
			IF (_cbEntrySize) > 0 THEN
				(* check index *)
				IF (_iEntry > 2) THEN
					(* error, too many entries *)
					nErrorId := BACnet_ERR_ADS_TooManyEntries;
					_i := 100;
				ELSE
					(* try to decode property data *)
					_strExtDecode(
						pChrStringExt:= ADR(_pEntry^.extString),
						cbOutSize	:= SIZEOF(arrTexts[_iEntry]),
						pOutString	:= ADR(arrTexts[_iEntry]),
						bValid		=> ,
						bOverflow	=> ,
						bUnsupported=> ,
						nLength		=> ,
						eSrcEncoding=> );
					(* check error flags *)
					IF _strExtDecode.bOverflow THEN
						(* text too long *)
						nErrorId := BACnet_ERR_ADS_WrongEntrySize;
						_i := 100;
					ELSIF _strExtDecode.bUnsupported THEN
						(* unsupported encoding *)
						nErrorId := BACnet_ERR_ADS_Encoding;
						_i := 100;
					END_IF
				END_IF
			END_IF

			(* next entry *)
			_NextEntry();
			_iEntry := _iEntry + 1;

			(* check if next entry available *)
			IF (NOT _bNextEntry) THEN
				IF (_iEntry < 3) THEN
					(* not enough entries *)
					nErrorId := BACnet_ERR_ADS_NotEnoughEntries;
				END_IF
				_i := 100;
			END_IF

		END_WHILE

	100: (* Done *)
		bDone := (nErrorId = BACnet_ERR_NO_ERROR);
		(* release ADS buffer *)
		stBACnet_AdsBuffer.iLocked := 0;
		(* go idle *)
		_i := 0;

END_CASE

(* set error flag *)
bError 	:= nErrorId > BACnet_ERR_NO_ERROR;
bBusy 	:= _i > 0;
END_FUNCTION_BLOCK
ACTION _NextEntry:
_bNextEntry := (_pEntry^.nEntrySize AND 16#80000000) = 16#80000000;
_cbTmpSize := _F_BACnet_AlignedSize((_pEntry^.nEntrySize AND 16#7FFFFFFF) + SIZEOF(_pEntry^.nEntrySize) + SIZEOF(_pEntry^.hdrInfo));
_pEntry := _pEntry + _cbTmpSize;
END_ACTION

(* POU FB_BACnet_ExceptionScheduleProperty, ST *)
FUNCTION_BLOCK FB_BACnet_ExceptionScheduleProperty
VAR_INPUT
	tObjectID			: T_BACnet_ObjectIdentifier := 16#FFFFFFFF;
	bAutoGet			: BOOL:=TRUE; (* TRUE = get data from property when ADS connection OR object ID changed *)
	bGet				: BOOL; (* FALSE --> TRUE = get data from property *)
	bSet				: BOOL; (* FALSE --> TRUE = set data into property *)
END_VAR
VAR_IN_OUT
	stExceptSched		: ST_BACnet_ExceptionScheduleBool;
	stAdsConn			: ST_BACnet_AdsConnection;
END_VAR
VAR_OUTPUT
	bDone				: BOOL;
	bBusy				: BOOL;
	bError				: BOOL;
	nErrorId			: UINT;
END_VAR
VAR
	_fbReadProp		: FB_BACnet_ReadProp;
	_fbWriteProp	: FB_BACnet_WriteProp;
	_i				: INT;
	_rtrigGet		: R_TRIG;
	_rtrigSet		: R_TRIG;

	_pOldEventEntrySize		: POINTER TO DWORD;
	_pSpEventCalEntryDate	: POINTER TO ST_BACnet_SpecialEventListCalEntryDate;
	_pSpEventCalEntryRange	: POINTER TO ST_BACnet_SpecialEventListCalEntryRange;
	_pSpEventCalEntryWnD	: POINTER TO ST_BACnet_SpecialEventListCalEntryWnD;
	_pSpEventCalRef			: POINTER TO ST_BACnet_SpecialEventListCalReference;
	_pTimeValue		: POINTER TO ST_BACnet_TimeValueList;
	_pOldTimeValue	: POINTER TO ST_BACnet_TimeValueList;

	_iEntry			: INT;
	_iTv			: INT;

	_bNextEvent		: BOOL;
	_bNextTimeValue	: BOOL;

	_cbTmpSize		: UDINT;
	_cbTotalEntry	: UDINT;
	_cbTotalBuf		: UDINT;
	_nAdsReloadOld	: USINT;
	_tObjectIDOld	: T_BACnet_ObjectIdentifier := 16#FFFFFFFF;

END_VAR
(*

Listheader:

typedef struct _ListEntryHdr
{
      DWORD nEntrySize;
      DWORD hdrInfo;
}ListEntryHdr, *PListEntryHdr;

#define ListAlignedSize(n)         (4*(((n)+3)/4))
#define FirstListEntry(p) ( (p)->nEntrySize == 0 )                          ? NULL:p
#define NextListEntry(p) ( ( ((p)->nEntrySize&0x80000000) == 0 ) ? NULL:(PBYTE)(p) + ( ListAlignedSize((p)->nEntrySize&~(0x80000000)) + sizeof(ListEntryHdr)) ) // +4 da für nEntrySize 4 Byte reserviert sind, HighBit ausmaskieren
#define ElemSize(p) ((p)->nEntrySize&(~0x80000000))
#define AlignedEntrySize(p) (ListAlignedSize((p)->nEntrySize&(~0x80000000)))

###################################################################

PropExceptionSchedule:

enum BACnetSpecialEventChoice
{
      calendarEntry,
      calendarReference,
      MaxBACnetSpecialEventChoice
};

typedef struct _BACnetCalendarEntry
{
      BACnetCalendarEntryChoice choice;
      union
      {
            BACnetDate              date;
            BACnetDateRange   dateRange;
            BACnetWeekNDay          weekNDay;
      };
}BACnetCalendarEntry, *PBACnetCalendarEntry;

enum BACnetValueChoice
{
      NullValue                    = 0,
      BoolValue                    = 1,
      UnsignedValue                = 2,
      SignedValue                  = 3,
      RealValue                    = 4,
      DoubleValue                  = 5,
      OctedStringValue        = 6,
      CharStringValue         = 7,
      ObjectIdentifierValue = 8,   // but DataType is 0x0C
      EnumerationValue        = 9,
      MaxBACnetValueChoice    = 10
};

typedef struct _BACnetValue  
{
      BACnetValueChoice choice;
      DWORD                        length;     // Alignment + Datenlänge die folgt
      union
      {
            BOOL                                     boolValue;
            FLOAT                                    realValue;
            DOUBLE                                   doubleValue;
            INT                                      signedValue;
            UINT                                     unsignedValue;
            BYTE*                                    pOctedStringValue; 
            CHAR*                                    pCharStringValue;
            BACnetObjectIdentifier  objectIdentifierValue;
            EnumerationValueType         enumerationValue;
      };
}BACnetValue, *PBACnetValue;

typedef struct _BACnetTimeValue
{
      BACnetTime time;
      DWORD  reserved;  // 64bit Alignment
      BACnetValue value;
}BACnetTimeValue, *PBACnetTimeValue;

typedef struct _BACnetTimeValueList
{
      DWORD nEntrySize; // 0x80000000 -> next entry
      DWORD reserved;
      BACnetTimeValue listEntry;
}BACnetTimeValueList, *PBACnetTimeValueList;

typedef struct _BACnetSpecialEvent
{
      BACnetSpecialEventChoice choice;
      union
      {
            BACnetCalendarEntry calendarEntry;
            BACnetObjectIdentifier calendarReference;
      };
      DWORD eventPriority; // DWORD due to alignment
      DWORD reserved;
      BACnetTimeValueList listOfTimeValues;
}BACnetSpecialEvent, *PBACnetSpecialEvent;

typedef struct _BACnetSpecialEventList
{
      DWORD nEntrySize; // 0x80000000 -> next entry
      DWORD reserved;
      BACnetSpecialEvent listEntry;
}BACnetSpecialEventList, *PBACnetSpecialEventList;

###################################################################

PropWeeklySchedule:

typedef struct _BACnetDailySchedule
{
      DWORD nEntrySize; // 0x80000000 -> next entry
      DWORD reserved;
      BACnetTimeValueList listEntry;
} BACnetDailySchedule, *PBACnetDailySchedule;

###################################################################

PropScheduleDefault / PropPresentValue

typedef struct _BACnetValueList
{
      DWORD nEntrySize; // 0x80000000 -> next entry
      DWORD reserved;
      BACnetValue listEntry;
} BACnetValueList, *PBACnetValueList;

###################################################################

*)

(* ADS read *)
_fbReadProp(
	BACnetDevicePort	:= stAdsConn.nAmsPort,
	bExecute			:= ,
	sNetId				:= stAdsConn.sAmsNetId,
	ObjectType			:= F_BACnet_GetObjType(tObjectID),
	PropertyID			:= BACnetPropertyIdentifier_ExceptionSchedule,
	DataType			:= BACnetDataType_SpecialEventList,
	ObjectInstance		:= F_BACnet_GetObjInstance(tObjectID),
	ptrValue			:= ADR(stBACnet_AdsBuffer.arrData),
	nLenValue			:= SIZEOF(stBACnet_AdsBuffer.arrData),
	bDone				=> ,
	bBusy				=> ,
	bError				=> ,
	nErrID				=> ,
	nProcessedLen		=> );

(* ADS write *)
_fbWriteProp(
	BACnetDevicePort	:= stAdsConn.nAmsPort,
	bExecute			:= ,
	sNetId				:= stAdsConn.sAmsNetId,
	ObjectType			:= F_BACnet_GetObjType(tObjectID),
	PropertyID			:= BACnetPropertyIdentifier_ExceptionSchedule,
	Priority			:= BACnetPriority_None,
	DataType			:= BACnetDataType_SpecialEventList,
	ObjectInstance		:= F_BACnet_GetObjInstance(tObjectID),
	ptrValue			:= ADR(stBACnet_AdsBuffer.arrData),
	nLenValue			:= _cbTotalBuf,
	bDone				=> ,
	bBusy				=> ,
	bError				=> ,
	nErrID				=> );

(* trigger start event *)
_rtrigGet(CLK:= bGet, Q=> );
_rtrigSet(CLK:= bSet, Q=> );

(* state machine *)
CASE _i OF

	0: (* Idle *)
		IF 		_rtrigGet.Q
			OR	_rtrigSet.Q
			OR	(		(		(_nAdsReloadOld <> stAdsConn.nReload)
							OR	(_tObjectIDOld <> tObjectID)
						)
					AND	bAutoGet
				)
			OR	stExceptSched.bReqGet
			OR	stExceptSched.bReqSet
		THEN
			IF (NOT stAdsConn.bValid) THEN
				(* ADS connection not valid *)
				nErrorId := BACnet_ERR_INVALID_ADS_CONN;
			ELSIF (NOT stAdsConn.bServer AND NOT stAdsConn.bClient) THEN
				(* not a server nor a client *)
				nErrorId := BACnet_ERR_ADS_NoServerClient;
			ELSE
				(* decide get or set *)
				IF _rtrigGet.Q OR stExceptSched.bReqGet  THEN
					_i := 1;
					stExceptSched.bReqGet := FALSE;
				ELSIF _rtrigSet.Q OR stExceptSched.bReqSet THEN
					_i := 11;
					stExceptSched.bReqSet := FALSE;
				ELSIF bAutoGet THEN
					_i := 1;
					stExceptSched.bReqGet := FALSE;
				END_IF
				nErrorId := BACnet_ERR_NO_ERROR;
				(* reset index *)
				_iEntry		:= 0;
				(* remind parameter *)
				_tObjectIDOld := tObjectID;
				_nAdsReloadOld := stAdsConn.nReload;
				(* lock data array *)
				stExceptSched.bBusy := TRUE;
			END_IF
			(* reset done flag *)
			bDone := FALSE;
		END_IF
		IF (NOT bGet) AND (NOT bSet) AND (NOT bAutoGet) THEN
			nErrorId := BACnet_ERR_NO_ERROR;
			bDone := FALSE;
		END_IF

	(* READ *)
	1: (* read object property data via ADS *)
		IF TestAndSet(stBACnet_AdsBuffer.bTestSet) THEN
			IF _fbReadProp.bExecute THEN
				IF _fbReadProp.bError THEN
					_i := 100;
					nErrorId := BACnet_ERR_ADS_Read;
					_fbReadProp.bExecute := FALSE;
				ELSIF (NOT _fbReadProp.bBusy) THEN
					_i := 2;
					_fbReadProp.bExecute := FALSE;
					(* prepare pointer *)
					_pSpEventCalEntryDate	:= ADR(stBACnet_AdsBuffer.arrData);
					_pSpEventCalEntryRange	:= ADR(stBACnet_AdsBuffer.arrData);
					_pSpEventCalEntryWnD	:= ADR(stBACnet_AdsBuffer.arrData);
					_pSpEventCalRef			:= ADR(stBACnet_AdsBuffer.arrData);
					(* clear output data *)
					MEMSET(ADR(stExceptSched.arrEntries), 0, SIZEOF(stExceptSched.arrEntries));
					_cbTotalBuf := 0;
					_bNextEvent := TRUE;
				END_IF

			ELSIF (stBACnet_AdsBuffer.iLocked = 0) THEN
				_fbReadProp.bExecute := TRUE;
				(* lock global ADS buffer *)
				stBACnet_AdsBuffer.iLocked := SIZEOF(stBACnet_AdsBuffer.arrData);
			END_IF

			(* release temporary task lock *)
			stBACnet_AdsBuffer.bTestSet := FALSE;
		END_IF

	2: (* select event entry *)
		(* more events? *)
		IF (NOT _bNextEvent) THEN
			(* no more events, exit *)
			_i := 4;
		ELSE
			_i := 3;
			(* check if local buffer is full *)
			IF _iEntry > BACnet_MaxExSchEntries THEN
				_i := 4; (* maximum entries reached --> finished *)
			ELSIF ((_pSpEventCalEntryDate^.nEntrySize AND 16#7FFFFFFF) > 0) THEN
				(* initialize first entry *)
				stExceptSched.arrEntries[_iEntry].eEntryType := BACnetCalendarEntryType_None;

				CASE _pSpEventCalEntryDate^.stListEntry.eEventChoice OF

					BACnetSpecialEventChoice_calendarReference:
						_pTimeValue := ADR(_pSpEventCalRef^.stListEntry.stListOfTimeValues);
						stExceptSched.arrEntries[_iEntry].eEntryType := BACnetCalendarEntryType_Ref;
						stExceptSched.arrEntries[_iEntry].stCalRef.tCalObjectId := _pSpEventCalRef^.stListEntry.tCalRef;
						stExceptSched.arrEntries[_iEntry].ePriority := DWORD_TO_INT(_pSpEventCalRef^.stListEntry.iEventPriority);

					BACnetSpecialEventChoice_calendarEntry:
						CASE _pSpEventCalEntryDate^.stListEntry.stCalEntry.eEntryChoice OF
							BACnetCalendarEntryChoice_date:
								_pTimeValue := ADR(_pSpEventCalEntryDate^.stListEntry.stListOfTimeValues);
								stExceptSched.arrEntries[_iEntry].eEntryType := BACnetCalendarEntryType_Date;
								stExceptSched.arrEntries[_iEntry].stDate.stStart := _pSpEventCalEntryDate^.stListEntry.stCalEntry.stDate;
								stExceptSched.arrEntries[_iEntry].stDate.stEnd := _pSpEventCalEntryDate^.stListEntry.stCalEntry.stDate;
								stExceptSched.arrEntries[_iEntry].ePriority := DWORD_TO_INT(_pSpEventCalEntryDate^.stListEntry.iEventPriority);

							BACnetCalendarEntryChoice_dateRange:
								_pTimeValue := ADR(_pSpEventCalEntryRange^.stListEntry.stListOfTimeValues);
								stExceptSched.arrEntries[_iEntry].eEntryType := BACnetCalendarEntryType_DateRange;
								stExceptSched.arrEntries[_iEntry].stDate.stStart := _pSpEventCalEntryRange^.stListEntry.stCalEntry.stStartDate;
								stExceptSched.arrEntries[_iEntry].stDate.stEnd := _pSpEventCalEntryRange^.stListEntry.stCalEntry.stEndDate;
								stExceptSched.arrEntries[_iEntry].ePriority := DWORD_TO_INT(_pSpEventCalEntryRange^.stListEntry.iEventPriority);

							BACnetCalendarEntryChoice_weekNDay:
								_pTimeValue := ADR(_pSpEventCalEntryWnD^.stListEntry.stListOfTimeValues);
								stExceptSched.arrEntries[_iEntry].eEntryType := BACnetCalendarEntryType_WeekNDay;
								stExceptSched.arrEntries[_iEntry].stWeekNDay.iMonth := _pSpEventCalEntryWnD^.stListEntry.stCalEntry.iMonth;
								stExceptSched.arrEntries[_iEntry].stWeekNDay.iWeekOfMonth := _pSpEventCalEntryWnD^.stListEntry.stCalEntry.iWeekOfMonth;
								stExceptSched.arrEntries[_iEntry].stWeekNDay.iDay := _pSpEventCalEntryWnD^.stListEntry.stCalEntry.iDay;
								stExceptSched.arrEntries[_iEntry].ePriority := DWORD_TO_INT(_pSpEventCalEntryWnD^.stListEntry.iEventPriority);

							ELSE
								(* unknown entry choice *)
								nErrorId := BACnet_ERR_UnknownEntryChoice;
								_i := 100;
						END_CASE
					ELSE
						(* unknown event choice *)
						nErrorId := BACnet_ERR_UnknownEventChoice;
						_i := 100;
				END_CASE
			ELSE
				(* mark as invalid *)
				stExceptSched.arrEntries[_iEntry].eEntryType := BACnetCalendarEntryType_None;
			END_IF
		END_IF
		(* reset time value index *)
		_iTv := 0;

	3: (* scan time value list *)
		(* preset next time value flag *)
		_bNextTimeValue := TRUE;
		(* loop till all time values are parsed *)
		WHILE _bNextTimeValue AND _pTimeValue <> 0 DO
			IF ((_pTimeValue^.nEntrySize AND 16#7FFFFFFF) > 0) AND (_iTv <= BACnet_MaxTimeValues) THEN
				(* time value data available - is it a bool type? *)
				IF		_pTimeValue^.stListEntry.stValue.eValueChoice = BACnetDataType_Bool
					OR	_pTimeValue^.stListEntry.stValue.eValueChoice = BACnetDataType_Null
				THEN
					(* decide entry type *)
					CASE stExceptSched.arrEntries[_iEntry].eEntryType OF
						BACnetCalendarEntryType_Date,
						BACnetCalendarEntryType_DateRange:
							stExceptSched.arrEntries[_iEntry].arrTimeValue[_iTv].bValid := TRUE;
							stExceptSched.arrEntries[_iEntry].arrTimeValue[_iTv].stTime := _pTimeValue^.stListEntry.stTime;
							stExceptSched.arrEntries[_iEntry].arrTimeValue[_iTv].eType := _pTimeValue^.stListEntry.stValue.eValueChoice;
							IF _pTimeValue^.stListEntry.stValue.cbData = 1 THEN
								MEMCPY(	ADR(stExceptSched.arrEntries[_iEntry].arrTimeValue[_iTv].bValue),
										ADR(_pTimeValue^.stListEntry.stValue.nData),
										SIZEOF(stExceptSched.arrEntries[_iEntry].arrTimeValue[_iTv].bValue)
								);
							ELSE
								stExceptSched.arrEntries[_iEntry].arrTimeValue[_iTv].bValue := FALSE;
							END_IF
							_iTv := _iTv +1;

						BACnetCalendarEntryType_WeekNDay:
							stExceptSched.arrEntries[_iEntry].arrTimeValue[_iTv].bValid := TRUE;
							stExceptSched.arrEntries[_iEntry].arrTimeValue[_iTv].stTime := _pTimeValue^.stListEntry.stTime;
							stExceptSched.arrEntries[_iEntry].arrTimeValue[_iTv].eType := _pTimeValue^.stListEntry.stValue.eValueChoice;
							IF _pTimeValue^.stListEntry.stValue.cbData = 1 THEN
								MEMCPY(	ADR(stExceptSched.arrEntries[_iEntry].arrTimeValue[_iTv].bValue),
										ADR(_pTimeValue^.stListEntry.stValue.nData),
										SIZEOF(stExceptSched.arrEntries[_iEntry].arrTimeValue[_iTv].bValue)
								);
							ELSE
								stExceptSched.arrEntries[_iEntry].arrTimeValue[_iTv].bValue := FALSE;
							END_IF
							_iTv := _iTv +1;

						BACnetCalendarEntryType_Ref:
							stExceptSched.arrEntries[_iEntry].arrTimeValue[_iTv].bValid := TRUE;
							stExceptSched.arrEntries[_iEntry].arrTimeValue[_iTv].stTime := _pTimeValue^.stListEntry.stTime;
							stExceptSched.arrEntries[_iEntry].arrTimeValue[_iTv].eType := _pTimeValue^.stListEntry.stValue.eValueChoice;
							IF _pTimeValue^.stListEntry.stValue.cbData = 1 THEN
								MEMCPY(	ADR(stExceptSched.arrEntries[_iEntry].arrTimeValue[_iTv].bValue),
										ADR(_pTimeValue^.stListEntry.stValue.nData),
										SIZEOF(stExceptSched.arrEntries[_iEntry].arrTimeValue[_iTv].bValue)
								);
							ELSE
								stExceptSched.arrEntries[_iEntry].arrTimeValue[_iTv].bValue := FALSE;
							END_IF
							_iTv := _iTv +1;

					END_CASE

				ELSE
					(* unsupported data type *);
				END_IF

			END_IF

			(* empty entry size or data buffer full, next time value entry *)
			_NextTimeValue();

		END_WHILE

		(* count *)(*
		IF _iTv > 0 THEN
			_iEntry := _iEntry +1;
		END_IF*)
		_iEntry := _iEntry +1;

		(* next event entry *)
		_NextEvent();
		_i := 2;

	4: (* data read and parsed successful *)
		stExceptSched.nGet := stExceptSched.nGet +1;
		_i := 100;

	11: (* lock global ADS buffer *)
		IF TestAndSet(stBACnet_AdsBuffer.bTestSet) THEN
			IF stBACnet_AdsBuffer.iLocked = 0 THEN
				stBACnet_AdsBuffer.iLocked := SIZEOF(stBACnet_AdsBuffer.arrData);
				(* initalize total size counter *)
				_cbTotalBuf := 0;
				(* prepare pointer *)
				_pSpEventCalEntryDate	:= ADR(stBACnet_AdsBuffer.arrData);
				_pSpEventCalEntryRange	:= ADR(stBACnet_AdsBuffer.arrData);
				_pSpEventCalEntryWnD	:= ADR(stBACnet_AdsBuffer.arrData);
				_pSpEventCalRef			:= ADR(stBACnet_AdsBuffer.arrData);
				_pOldEventEntrySize		:= 0;
				(* loop against input data *)
				_i := 12;
			END_IF
			(* release temporary task lock *)
			stBACnet_AdsBuffer.bTestSet := FALSE;
		END_IF

	12: (* write calendar entries date/date range *)
		FOR _iEntry := 0 TO BACnet_MaxExSchEntries DO

			_pOldTimeValue	:= 0;
			_cbTotalEntry	:= 0;

			IF stExceptSched.arrEntries[_iEntry].eEntryType <> BACnetCalendarEntryType_None THEN
				(* valid entry *)
				CASE stExceptSched.arrEntries[_iEntry].eEntryType OF

					BACnetCalendarEntryType_Date,
					BACnetCalendarEntryType_DateRange:
						(* set special entry choice *)
						IF stExceptSched.arrEntries[_iEntry].eEntryType = BACnetCalendarEntryType_Date THEN
							_pSpEventCalEntryDate^.stListEntry.eEventChoice := BACnetSpecialEventChoice_calendarEntry;
							_pSpEventCalEntryDate^.stListEntry.nRes1 := 0;
							(* set time value pointer *)
							_pTimeValue := ADR(_pSpEventCalEntryDate^.stListEntry.stListOfTimeValues);
						ELSE
							_pSpEventCalEntryRange^.stListEntry.eEventChoice := BACnetSpecialEventChoice_calendarEntry;
							_pSpEventCalEntryRange^.stListEntry.nRes1 := 0;
							(* set time value pointer *)
							_pTimeValue := ADR(_pSpEventCalEntryRange^.stListEntry.stListOfTimeValues);
						END_IF

					BACnetCalendarEntryType_WeekNDay:
						(* set special entry choice *)
						_pSpEventCalEntryWnD^.stListEntry.eEventChoice := BACnetSpecialEventChoice_calendarEntry;
						_pSpEventCalEntryWnD^.stListEntry.nRes1 := 0;
						(* set time value pointer *)
						_pTimeValue := ADR(_pSpEventCalEntryWnD^.stListEntry.stListOfTimeValues);

					BACnetCalendarEntryType_Ref:
						(* set special entry choice *)
						_pSpEventCalRef^.stListEntry.eEventChoice := BACnetSpecialEventChoice_calendarReference;
						_pSpEventCalRef^.stListEntry.nRes1 := 0;
						(* set time value pointer *)
						_pTimeValue := ADR(_pSpEventCalRef^.stListEntry.stListOfTimeValues);

				END_CASE


				(* loop against time values *)
				FOR _iTv := 0 TO BACnet_MaxTimeValues DO

					(* valid entry? *)
					IF stExceptSched.arrEntries[_iEntry].arrTimeValue[_iTv].bValid THEN
						(* copy time *)
						_pTimeValue^.stListEntry.stTime := stExceptSched.arrEntries[_iEntry].arrTimeValue[_iTv].stTime;
						_pTimeValue^.stListEntry.stValue.nData := 0; (* clear data *)
						(* decide between None and Bool type *)
						IF stExceptSched.arrEntries[_iEntry].arrTimeValue[_iTv].eType = BACnetDataType_Bool THEN
							(* BOOL type *)
							_pTimeValue^.stListEntry.stValue.eValueChoice := BACnetDataType_Bool;
							_pTimeValue^.stListEntry.stValue.nRes1 := 0;
							_pTimeValue^.stListEntry.stValue.cbData := SIZEOF(stExceptSched.arrEntries[_iEntry].arrTimeValue[_iTv].bValue);
							MEMCPY(	ADR(_pTimeValue^.stListEntry.stValue.nData),
									ADR(stExceptSched.arrEntries[_iEntry].arrTimeValue[_iTv].bValue),
									MIN(SIZEOF(_pTimeValue^.stListEntry.stValue.nData), _pTimeValue^.stListEntry.stValue.cbData)
							);
						ELSE
							(* other or NONE type *)
							_pTimeValue^.stListEntry.stValue.eValueChoice := BACnetDataType_Null;
							_pTimeValue^.stListEntry.stValue.nRes1 := 0;
							_pTimeValue^.stListEntry.stValue.cbData := 0;
						END_IF

						(* calculate time-value entry size *)
						_pTimeValue^.nEntrySize :=	_pTimeValue^.stListEntry.stValue.cbData
												+	SIZEOF(_pTimeValue^.stListEntry.nRes)
												+	SIZEOF(_pTimeValue^.stListEntry.stTime)
												+	SIZEOF(_pTimeValue^.stListEntry.stValue.cbData)
												+	SIZEOF(_pTimeValue^.stListEntry.stValue.eValueChoice)
												+	SIZEOF(_pTimeValue^.stListEntry.stValue.nRes1);

						IF (_iTv > 0 AND _pOldTimeValue <> 0) THEN
							(* next entry flag *)
							_pOldTimeValue^.nEntrySize := _pOldTimeValue^.nEntrySize + 16#80000000;
						END_IF

						(* update time value pointer *)
						_NextTimeValue();

						(* ...and add to total entry size counter *)
						_cbTotalEntry := _cbTotalEntry + _cbTmpSize;

					ELSE
						(* clear entry *)
						_pTimeValue^.nEntrySize := 0;
						_pTimeValue^.stListEntry.stValue.cbData := 0;
					END_IF

				END_FOR

				(* check if time value list is empty *)
				IF _cbTotalEntry = 0 THEN
					(* no time values, set default size *)
					_cbTotalEntry := SIZEOF(_pTimeValue^.nEntrySize) + SIZEOF(_pTimeValue^.nRes);
				END_IF

				(* caclulate event entry size *)
				CASE stExceptSched.arrEntries[_iEntry].eEntryType OF

					BACnetCalendarEntryType_Date:
						(* caclulate event entry size and write into data structure *)
						_pSpEventCalEntryDate^.nEntrySize :=	_cbTotalEntry
															+	SIZEOF(_pSpEventCalEntryDate^.stListEntry.eEventChoice)
															+	SIZEOF(_pSpEventCalEntryDate^.stListEntry.iEventPriority)
															+	SIZEOF(_pSpEventCalEntryDate^.stListEntry.nRes1)
															+	SIZEOF(_pSpEventCalEntryDate^.stListEntry.nRes2)
															+	SIZEOF(_pSpEventCalEntryDate^.stListEntry.nRes3)
															+	SIZEOF(_pSpEventCalEntryDate^.stListEntry.stCalEntry);
						(* copy event data *)
						_pSpEventCalEntryDate^.stListEntry.eEventChoice := BACnetSpecialEventChoice_calendarEntry;
						_pSpEventCalEntryDate^.stListEntry.nRes1 := 0;
						_pSpEventCalEntryDate^.stListEntry.iEventPriority := stExceptSched.arrEntries[_iEntry].ePriority;
						_pSpEventCalEntryDate^.stListEntry.stCalEntry.eEntryChoice := BACnetCalendarEntryChoice_date;
						_pSpEventCalEntryDate^.stListEntry.stCalEntry.nRes := 0;
						_pSpEventCalEntryDate^.stListEntry.stCalEntry.stDate := stExceptSched.arrEntries[_iEntry].stDate.stStart;

